	20:	// Oczekiwanie na zapis statusu - sprawdzenie wyniku
		IF stStationSettings.bSkipCheckStatusSaveResult THEN
			fbLogger.mAppendCurrentLine(bBreakLine := FALSE, sAddSep := '', sAppendText:= ', CSSR_Skiped');	
			IF bLastStatus THEN
				iCtr_PIM_PartsOK := iCtr_PIM_PartsOK +1;
			ELSE
				iCtr_PIM_PartsNOK := iCtr_PIM_PartsNOK +1;
			END_IF
			iWorkStep := 25;			
		ELSIF NOT bInsertStatus THEN
			IF bStatusSavedOK THEN
				IF bLastStatus THEN
					iCtr_PIM_PartsOK := iCtr_PIM_PartsOK +1;
				ELSE
					iCtr_PIM_PartsNOK := iCtr_PIM_PartsNOK +1;
				END_IF
				fbLogger.mAppendCurrentLine(bBreakLine := FALSE, sAddSep := '', sAppendText:= ', StatusSaved');
				iWorkStep := 25;	
			ELSE
				fbLogger.mAppendCurrentLine(bBreakLine := FALSE, sAddSep := '', sAppendText:= ', StatusNotSaved');
				mNewEvent(nInputErrorID := nPIM_ErrorCodes.StatusSaveError, nEventType := nPIM_EventClasses.Alarm, tMessageTime := T#0S);
			END_IF
		END_IF
		
	25:	// Oczekiwanie na zakończenie operacji
		IF NOT bSaveStatus THEN 
			fbLogger.mAppendCurrentLine(bBreakLine := TRUE, sAddSep := '', sAppendText:= ', OperEnded_BaseState_2');
			bNewOperationInProgress := FALSE;
			iWorkStep := 10;	
		END_IF

	99:
		IF stPimInOut.bConfirmEvent AND stPimInOut.bPIMActive THEN
			bResetSignal := TRUE;
			fbLogger.mAddLine(sTextToSave := CONCAT(STR1:= 'Reset bledu - wewnetrznego', STR2:= stPimInOut.sErrorCodePLC ) );
			IF 	nErrorID = nPIM_ErrorCodes.SelectStationIdError THEN 		// Błąd w inicjalizacji stanowiska do pracy
				nErrorID := nPIM_ErrorCodes.NoError;
				iWorkStep := 0;
			ELSIF nErrorID = nPIM_ErrorCodes.StatusSaveError THEN			// Gdy błąd zapisu statusu spróbuj jeszcze raz
				nErrorID := nPIM_ErrorCodes.NoError;
				bInsertStatus := TRUE;
				iWorkStep := 20;
			ELSE
				nErrorID := nPIM_ErrorCodes.NoError;
				iWorkStep := 0;
			END_IF
			IF nErrorID = nPIM_ErrorCodes.NoError THEN	// Jeśli błąd potwierdzony
				stPimInOut.bNonBlockingAlarm := stPimInOut.bAlarmPLC := stPimInOut.bWorkBlock_PLC := FALSE;
				stPimInOut.sErrorCodePLC := '';
				bResetSignal := FALSE;
				nEventType := nPIM_EventClasses.NoError;
			END_IF
		ELSIF nEventType = nPIM_EventClasses.Message THEN
				iWorkStep := 10;
		ELSE
			IF (nEventType <>nPIM_EventClasses.NoError) AND (NOT stPimInOut.bAlarmPLC AND NOT stPimInOut.bWorkBlock_PLC)  THEN
				mNewEvent(nInputErrorID := nPIM_ErrorCodes.UnKnownAlarm, nEventType := nPIM_EventClasses.Error, tMessageTime := T#0S);	
			END_IF
		END_IF
	
END_CASE

ACT_PimCmdsHandling();		// Obsługa komend z/do PIMu
ACT_SqlDataReturnCmd();		// Obsługa zapytań SQL do DB


// Automatyczne kasowanie wiadomości po zadanym czasie wyświetlania lub alarmu przy starcie nowej operacji
fbTON_MessageTimer();
IF stPimInOut.bNonBlockingAlarm AND (fbTON_MessageTimer.Q OR nMachineState = nPIM_MachineStates._3_NewOperationStarted) THEN
	fbTON_MessageTimer(IN:= FALSE);
	stPimInOut.sErrorCodePLC := '';
	stPimInOut.bNonBlockingAlarm := stPimInOut.bAlarmPLC := FALSE;
	nEventType := nPIM_EventClasses.NoError;
END_IF

fbTON_ServiceMessageTimer();		// Reset wiadomości serwisowej
IF fbTON_ServiceMessageTimer.Q THEN
	fbTON_ServiceMessageTimer(IN:= FALSE);
	stPimInOut.sPlcServiceMessage := '';
END_IF

IF GVL_Aircom.stAC_DT_Data.bNew_Shift OR bTestZapisu THEN
	iCtrMem_Operations := iCtr_Operations;
	iCtrMem_OperationsInterrupted := iCtr_OperationsInterrupted;
	iCtrMem_OperationsEndedOK := iCtr_OperationsEndedOK;
	iCtrMem_OperEndedOK_Method := iCtr_OperEndedOK_Method;
	iCtrMem_OperationsEndedNOK := iCtr_OperationsEndedNOK;
	iCtrMem_PIM_PartsOK := iCtr_PIM_PartsOK;
	iCtrMem_PIM_PartsNOK := iCtr_PIM_PartsNOK;
	iCtrMem_PIM_ReworkYes := iCtr_PIM_ReworkYes;
	iCtrMem_PIM_PartOK_SaveError := iCtr_PIM_PartOK_SaveError;
	iCtrMem_PIM_PartNOK_SaveError := iCtr_PIM_PartNOK_SaveError;
	iCtrMem_StatusSaveOK := iCtr_StatusSaveOK;
	iCtrMem_StatusSaveError := iCtr_StatusSaveError;
	iCtrMem_Errors := iCtr_Errors;
	iCtr_Operations:= iCtr_OperationsInterrupted:= iCtr_OperationsEndedOK:= iCtr_OperEndedOK_Method:= iCtr_OperationsEndedNOK:= 0; 
	iCtr_PIM_PartsOK:= iCtr_PIM_PartsNOK:= iCtr_PIM_ReworkYes:= iCtr_PIM_PartOK_SaveError := iCtr_PIM_PartNOK_SaveError:= iCtr_StatusSaveOK:= iCtr_StatusSaveError:= iCtr_Errors:= 0;

fbLogger.mAddLine(sTextToSave := CONCAT(STR1:= 'Nowa zmiana - ', STR2:= UINT_TO_STRING( GVL_Aircom.stAC_DT_Data.uiShiftNumber) ));
	fbLogger.mSaveBuffor();
	bTestZapisu := FALSE;
	bWriteHistoricData := TRUE;
END_IF
IF bWriteHistoricData AND fbLogger.bBufferEmpty THEN
		fbFormatStr(sFormat := 'PrevShiftReport: Oper-%d, OperInt-%d, OperOK-%d, OperOK_M-%d, OperNOK-%d',
		arg1 := F_INT(iCtrMem_Operations), 
		arg2 := F_INT(iCtrMem_OperationsInterrupted), 
		arg3 := F_INT(iCtrMem_OperationsEndedOK), 
		arg4 := F_INT(iCtrMem_OperEndedOK_Method), 
		arg5 := F_INT(iCtrMem_OperationsEndedNOK));  
	fbLogger.mAddLine(sTextToSave := fbFormatStr.sOut );
	fbFormatStr(sFormat := 'PrevShiftReport: PartsPIM_OK-%d, PartsPIM_NOK-%d, PartsPIM_ReworkYes-%d, PartsPIM_OK_missed-%d, PartsPIM_NOK_Missed-%d',
		arg1 := F_INT(iCtrMem_PIM_PartsOK), 
		arg2 := F_INT(iCtrMem_PIM_PartsNOK), 
		arg4 := F_INT(iCtrMem_PIM_ReworkYes),
		arg5 := F_INT(iCtrMem_PIM_PartOK_SaveError), 
		arg6 := F_INT(iCtrMem_PIM_PartNOK_SaveError));  
	fbLogger.mAddLine(sTextToSave := fbFormatStr.sOut );
	fbFormatStr(sFormat := 'PrevShiftReport: StatusSaveOK-%d, StatusSaveError-%d, Errors-%d, CmdReset- %d',
		arg1 := F_INT(iCtrMem_StatusSaveOK), 
		arg2 := F_INT(iCtrMem_StatusSaveError), 
		arg3 := F_INT(iCtrMem_Errors), 
		arg3 := F_UINT(in:=uiCtr_CmdReset));  
	uiCtr_CmdReset := 0;
	fbLogger.mAddLine(sTextToSave := fbFormatStr.sOut );	
	fbLogger.mSaveBuffor();
	bWriteHistoricData := FALSE;
END_IF

fbTON_ConfirmReset(IN:= stPimInOut.bConfirmEvent, PT:= T#3S);
stPimInOut.bConfirmEvent R= fbTON_ConfirmReset.Q;

PROPERTY PartsCtr_NOK : INT
GET
PartsCtr_NOK := iCtr_PIM_PartsNOK;
END_GET
END_PROPERTY

PROPERTY PartsCtr_OK : INT
GET
PartsCtr_OK := iCtr_PIM_PartsOK;
END_GET
END_PROPERTY

// The number of actually displayed error code ex "601"
PROPERTY prActiveErrorCode : STRING
GET
prActiveErrorCode := stPimInOut.sErrorCodePLC;
END_GET
END_PROPERTY

(* Get CMD Value from PIM*)
PROPERTY prCMD : STRING
GET
IF __ISVALIDREF(stPimInOut) THEN
	prCMD := sCmdToSendToMachine;
	sCmdToSendToMachine := '';	
END_IF
END_GET
END_PROPERTY

(* Get info *)
PROPERTY prCurrentMachineState : nPIM_MachineStates
GET
prCurrentMachineState := nMachineState;
END_GET
END_PROPERTY

(* Get info *)
PROPERTY prErrorClassExt : nPIM_EventClasses
GET
prErrorClassExt := nActEventClass;
END_GET
END_PROPERTY

(* Get info *)
PROPERTY prErrorConfirmActive : BOOL
GET
IF __ISVALIDREF(stPimInOut) THEN
	prErrorConfirmActive := stPimInOut.bConfirmEvent;
END_IF
END_GET
END_PROPERTY

(* Get info *)
PROPERTY prExternalEvtWaitInQueue : BOOL
GET
prExternalEvtWaitInQueue := FALSE;
END_GET
END_PROPERTY

(* Get info is PIM is active*)
PROPERTY prLastSavedStatus : BOOL
GET
prLastSavedStatus := bLastStatus;
END_GET
END_PROPERTY

(* Get info is PIM is active*)
PROPERTY prNokReportedSource : nPIM_ReportedNokSource
GET
prNokReportedSource := nReoprtedNokSource;
END_GET
END_PROPERTY

(* Get info is PIM is active*)
PROPERTY prOperEnded : BOOL
GET
prOperEnded := bOperationEnded;
END_GET
END_PROPERTY

(* Get info is PIM is active*)
PROPERTY prOperInProgress : BOOL
GET
prOperInProgress := nMachineState >= nPIM_MachineStates._3_NewOperationStarted AND nMachineState <= nPIM_MachineStates._6_ReturningToBaseState;
END_GET
END_PROPERTY

(* Get info is PIM is active*)
PROPERTY prPimActive : BOOL
GET
IF __ISVALIDREF(stPimInOut) THEN
	prPimActive := stPimInOut.bPIMActive;
END_IF
END_GET
END_PROPERTY

(* Get info *)
PROPERTY prPimBlockWork : BOOL
GET
IF __ISVALIDREF(stPimInOut) THEN
	prPimBlockWork := stPimInOut.bWorkBlock_PIM;
END_IF
END_GET
END_PROPERTY

(* Get info *)
PROPERTY prPlcBlockWork : BOOL
GET
IF __ISVALIDREF(stPimInOut) THEN
	prPlcBlockWork := stPimInOut.bWorkBlock_PLC;
END_IF
END_GET
END_PROPERTY

(* Get info is PIM is active*)
PROPERTY prReworkStatus : nPIM_ReworkSelect
GET
prReworkStatus := nReworkMenuStatus;
END_GET
END_PROPERTY

// Get info if station data is correctlly downloaded from database
PROPERTY prStationDataOK : BOOL
GET
prStationDataOK := bStationDataOK;
END_GET
END_PROPERTY

(* Get info is test mode is active*)
PROPERTY prTestMode : BOOL
GET
IF __ISVALIDREF(stPimInOut) THEN
	prTestMode := stPimInOut.bTestMode;
END_IF
END_GET
END_PROPERTY

(* Get info is user are logged?*)
PROPERTY prUserLogged : BOOL
GET
prUserLogged := fbTON_UserLogedDeleyed.Q;
END_GET
END_PROPERTY

(* Get info *)
PROPERTY prWorkPermission : BOOL
GET
IF __ISVALIDREF(stPimInOut) THEN
	prWorkPermission := stPimInOut.bTestMode OR NOT stPimInOut.bPIMActive OR (stPimInOut.bUSerLogged AND NOT stPimInOut.bWorkBlock_PIM AND NOT stPimInOut.bWorkBlock_PLC
					AND (NOT stPimInOut.bAlarmPLC OR stPimInOut.bNonBlockingAlarm) AND bMachineParamsOK AND bStationDataOK AND NOT bRetool AND NOT bMachParamsReadFromDB 
					AND NOT bMachParamsSendToDB);
END_IF
END_GET
END_PROPERTY

(* Get info is that machine is EOL*)
PROPERTY prIsEol : BOOL
GET
prIsEol := stRetDataLineStation.IsEOL;
END_GET
END_PROPERTY

(* Get Station name followed by machine number ex: 'CA01PL19_1'*)
PROPERTY prPartCodeNumber : STRING(250)
GET
prPartCodeNumber := stRetDataLineStation.PartCodeNumber;
END_GET
END_PROPERTY

(* Get Hidden status info*)
PROPERTY prIsHidden : BOOL
GET
prIsHidden := bIsHidden;
END_GET
END_PROPERTY

(* Get Line name ex: 'CA01PL'*)
PROPERTY prLineName : STRING(31)
GET
prLineName := sLineName;
END_GET
END_PROPERTY

(* Get Machine number*)
PROPERTY prMachNumber : INT
GET
prMachNumber := iMachineNumber;
END_GET
END_PROPERTY

(* Get Station name followed by machine number ex: 'CA01PL19_1'*)
PROPERTY prStationAlias : STRING(31)
GET
prStationAlias := CONCAT(STR1:= CONCAT(STR1:= sStationName, '_'), INT_TO_STRING(iMachineNumber));
END_GET
END_PROPERTY

(* Get Station name ex: 'CA01PL19'*)
PROPERTY prStationName : STRING(31)
GET
prStationName := sStationName;
END_GET
END_PROPERTY

// Zapis do DB dodatkowego kodu błędu - jeśli rozkaz dodany do kolejki zmienna wyjściowa ma wartość TRUE, jeśli nie (błąd dodania) FALSE
METHOD m_SqlInsAdditionalError : BOOL
VAR_INPUT
	sErrCode:STRING(10);		// Kod błędu do wysłania
END_VAR
VAR
	bResult:BOOL;
END_VAR
IF sErrCode <> '' AND stRetDataLineStation.IdStacji <> 0 THEN
	stSqlComandDataTMP.nCmdState:= nSQL_CmdExecState.New;
	stSqlComandDataTMP.nCmdType:=nSQL_CmdTypes.InsAdditionalError;
	stSqlComandDataTMP.bWaitForDataReturn:=FALSE;
	sFormat := 'INSERT INTO [dbo].[ProductionLineStationAdditionalError] (IdLineStation, MachineNumber, IdMachineError) VALUES (%d, %d, COALESCE( (SELECT Id FROM [dbo].[ProductionMachineError] WHERE Active = 1 AND Code = $'%s$'), -9223372036854775285))';
	fbFormatStr2(pFormatString := ADR(sFormat),
			arg1:= F_DINT(stRetDataLineStation.IdStacji),
			arg2:= F_INT(iMachineNumber),
			arg3:= F_STRINGEx(sErrCode),
			pDstString := ADR(stSqlComandDataTMP.sCmdExpression), nDstSize := SIZEOF(stSqlComandDataTMP.sCmdExpression));

	stSqlComandDataTMP.pReturnedData := 0;
	stSqlComandDataTMP.uiReturnedDataSize := 0;	
	IF I_SqlCore <> 0 THEN
		bResult := I_SqlCore.mAddCmdToQueue(ADR(stSqlComandDataTMP));
	END_IF
	m_SqlInsAdditionalError := bResult;
ELSE
	m_SqlInsAdditionalError := FALSE;
END_IF
END_METHOD

// Zapis do DB licznika zużycia powietrza - jeśli rozkaz dodany do kolejki zwraca TRUE, jeśli nie FALSE
METHOD m_SqlInsCompressedAirConsumption : BOOL
VAR_INPUT
	rActCompressedAirConsumption:REAL;		// Wartość licznika zużycia sprężonego powietrza
END_VAR
IF rActCompressedAirConsumption <> 0 AND stRetDataLineStation.IdLinii <> 0 THEN
	stSqlComandDataTMP.nCmdState:= nSQL_CmdExecState.New;
	stSqlComandDataTMP.nCmdType:=nSQL_CmdTypes.InsCompressedAirCons;
	stSqlComandDataTMP.bWaitForDataReturn:=FALSE;
	
	sFormat := 'INSERT INTO `ProductionConsumption_CompressedAir` (`IdLine`, `CounterValue`, `ValueUnit`) VALUES ( %d, %.3f, $'m3$')';
	fbFormatStr2(pFormatString := ADR(sFormat),
			arg1:= F_DINT(stRetDataLineStation.IdLinii),
			arg2:= F_REAL(rActCompressedAirConsumption),
			pDstString := ADR(stSqlComandDataTMP.sCmdExpression), nDstSize := SIZEOF(stSqlComandDataTMP.sCmdExpression));
	stSqlComandDataTMP.pReturnedData := 0;
	stSqlComandDataTMP.uiReturnedDataSize := 0;	
	IF I_SqlCore <> 0 THEN
		m_SqlInsCompressedAirConsumption := I_SqlCore.mAddCmdToQueue(ADR(stSqlComandDataTMP));
	END_IF	
ELSE
	m_SqlInsCompressedAirConsumption := FALSE;
END_IF
END_METHOD

// Zapis do DB relacji ostatniego statusu z kodem błędu - jeśli rozkaz dodany do kolejki zwraca TRUE, jeśli nie FALSE
METHOD m_SqlInsDefectRelation : BOOL
VAR_INPUT
	sErrCode:STRING(10);			// Kod błędu
END_VAR
IF sErrCode <> '' THEN
	stSqlComandDataTMP.nCmdState:= nSQL_CmdExecState.New;
	stSqlComandDataTMP.nCmdType:=nSQL_CmdTypes.InsDefectRelation;
	stSqlComandDataTMP.bWaitForDataReturn:=FALSE;
	
	sFormat := 'INSERT INTO [dbo].[ProductionMachinePartsStatusDefectRelation] (IdPartStatus, IdMachineError) values (%d, (SELECT Id FROM [dbo].[ProductionMachineError] WHERE Active = 1 AND Code = $'%s$'))';
	fbFormatStr2(pFormatString := ADR(sFormat),
			arg1:= F_LINT(liLPartStatusId),
			arg2:= F_STRINGEx(sErrCode),
			pDstString := ADR(stSqlComandDataTMP.sCmdExpression), nDstSize := SIZEOF(stSqlComandDataTMP.sCmdExpression));

	stSqlComandDataTMP.pReturnedData := 0;
	stSqlComandDataTMP.uiReturnedDataSize := 0;	
	IF I_SqlCore <> 0 THEN
		m_SqlInsDefectRelation := I_SqlCore.mAddCmdToQueue(ADR(stSqlComandDataTMP));
	END_IF
ELSE
	m_SqlInsDefectRelation := FALSE;
END_IF
END_METHOD

// Zapis do DB licznika zużycia energi na stanowisku - jeśli rozkaz dodany do kolejki zwraca TRUE, jeśli nie FALSE
METHOD m_SqlInsEnergyConsumption : BOOL
VAR_INPUT
	rActEnergyConsumption:REAL;			// Wartość licznika zużycia energii elektrycznej
END_VAR
IF rActEnergyConsumption <> 0 AND stRetDataLineStation.IdStacji <> 0 THEN
	stSqlComandDataTMP.nCmdState:= nSQL_CmdExecState.New;
	stSqlComandDataTMP.nCmdType:=nSQL_CmdTypes.InsEnergyCons;
	stSqlComandDataTMP.bWaitForDataReturn:=FALSE;
	
	sFormat := 'INSERT INTO `ProductionConsumption_Energy` (`IdLineStation`, `CounterValue`, `ValueUnit`) VALUES ( %d, %.3f, $'kWh$')';
	fbFormatStr2(pFormatString := ADR(sFormat),
			arg1:= F_DINT(stRetDataLineStation.IdStacji),
			arg2:= F_REAL(rActEnergyConsumption),
			pDstString := ADR(stSqlComandDataTMP.sCmdExpression), nDstSize := SIZEOF(stSqlComandDataTMP.sCmdExpression));

	stSqlComandDataTMP.pReturnedData := 0;
	stSqlComandDataTMP.uiReturnedDataSize := 0;	
	IF I_SqlCore <> 0 THEN
		m_SqlInsEnergyConsumption := I_SqlCore.mAddCmdToQueue(ADR(stSqlComandDataTMP));
	END_IF
ELSE
	m_SqlInsEnergyConsumption := FALSE;
END_IF
END_METHOD

// Zapis do DB danych rozszerzonych operacji - jeśli rozkaz dodany do kolejki zwraca TRUE, jeśli nie FALSE
METHOD m_SqlInsertExtendedData : BOOL		
VAR_INPUT
	pParameters: POINTER TO BYTE;				// Wskaźnik na tablicę elementów typu PIM_ExtDataRow
	uiArraySize: UINT;							// Rozmiar tablicy parametrów (może być pojedyncza zmienna)
END_VAR
VAR
	pExtData: POINTER TO stPIM_ExtDataRow;
	i:UINT;
	uiLastIndex:UINT;
END_VAR
uiLastIndex := uiArraySize/ SIZEOF(stPIM_ExtDataRow);
IF pParameters <> 0 AND uiArraySize > 0 AND uiLastIndex > 0 AND liLPartStatusId <> 0 THEN		// Zabezpieczenie przed brakiem danych wejściowych
	stSqlComandDataTMP.sCmdExpression := 'INSERT INTO `ProductionMachinePartParams` (`IdPartStatus`,`Name`,`Value`) VALUES';
	pExtData := pParameters;
	FOR i:=1 TO uiLastIndex DO		// Dodanie do stringa wartości
		IF i = uiLastIndex THEN		// Ostatnia wartość bez przecinka
			fbFormatStr(sFormat:= ' (%d,$'%s$',$'%s$')',arg1 := F_LINT(in:=liLPartStatusId), arg2 := F_STRINGEx(pExtData^.sName), arg3 := F_STRINGEx(pExtData^.sValue));
		ELSE
			fbFormatStr(sFormat:= ' (%d,$'%s$',$'%s$'),',arg1 := F_LINT(in:=liLPartStatusId), arg2 := F_STRINGEx(pExtData^.sName), arg3 := F_STRINGEx(pExtData^.sValue));		
			pExtData := pExtData + SIZEOF(stPIM_ExtDataRow);		// Przejście na kolejny indeks w tablicy
		END_IF
		CONCAT2(pSrcString1 := ADR(stSqlComandDataTMP.sCmdExpression), pSrcString2 := ADR(fbFormatStr.sOut), pDstString := ADR(stSqlComandDataTMP.sCmdExpression), nDstSize:= SIZEOF(stSqlComandDataTMP.sCmdExpression));
	END_FOR
	stSqlComandDataTMP.nCmdState:= nSQL_CmdExecState.New;
	stSqlComandDataTMP.nCmdType:=nSQL_CmdTypes.InsExtendedData;
	stSqlComandDataTMP.bWaitForDataReturn:=FALSE;
	stSqlComandDataTMP.pReturnedData := 0;
	stSqlComandDataTMP.uiReturnedDataSize := 0;
	IF I_SqlCore <> 0 THEN
  		m_SqlInsertExtendedData := I_SqlCore.mAddCmdToQueue(ADR(stSqlComandDataTMP));
	END_IF
ELSE
	m_SqlInsertExtendedData := FALSE;
END_IF
END_METHOD

// Zapis do DB parametrów maszyny przypisanych do aktualnego komponentu - gdy rozkaz zostanie wykonany zwraca TRUE
METHOD m_SqlInsMachineParamsData : BOOL
VAR_INPUT
	pParamsData: POINTER TO BYTE;		// Wskaźnik do bloku parametrów maszyny
	uiParamsDataSize: UINT;				// ROzmiar bloku danych parametrów maszyny
	wCrcSumOfParameters:WORD:= 0;
END_VAR
VAR_OUTPUT
	bProcessing:BOOL;					// Przetwarzanie rozkazu trwa (rozkaz dodany do kolejki)
	bResultOK:BOOL;						// Wynik wykonania rozkazu (do sprawdzenia gdy metoda zwróci TRUE)
	diParamsId:DINT;					// Id parametrów w DB
END_VAR
VAR
	sStringTMP:STRING(1000);
	iCRC16sum: INT;
END_VAR

// Sprawdzenie danych wejściowych - jeśli błędne przerwij procedure
IF pParamsData = 0 OR uiParamsDataSize = 0 OR stRetDataLineStation.IdStacji = 0 THEN 
	nErrorID:=nPIM_ErrorCodes.ProgramError;
	RETURN;
END_IF

// Rezerwacja struktury danych dla zapytania
IF NOT bReturnDataBusy OR bReturnDataReserved_InsMachParams THEN
	IF NOT bCmdSended THEN	// Przygotowanie danych do zapytania
		stSqlComandData.nCmdState:= nSQL_CmdExecState.New;
		stSqlComandData.nCmdType:=nSQL_CmdTypes.InsMachineParams;
		stSqlComandData.byExecutingNodeNb:=0;
		stSqlComandData.bWaitForDataReturn:=TRUE;
		
		IF wCrcSumOfParameters <> 0 THEN
			iCRC16sum := WORD_TO_INT(wCrcSumOfParameters);
		ELSE
			iCRC16sum := WORD_TO_INT(F_DATA_TO_CRC16_CCITT(pData := pParamsData, cbData := uiParamsDataSize, crc:= 0));
		END_IF
		
		sFormat := 'UPDATE [dbo].[ProductionMachineParameters] SET Active = 0 WHERE IdLineStation = %d AND MachineNumber = %d AND IdComposedPart = %d DECLARE @ID_INSERTED TABLE (Id INT) INSERT INTO [dbo].[ProductionMachineParameters] 
					(IdLineStation, MachineNumber, IdComposedPart,ParamsData,CRC_Sum,ParamsSizeInBytes) OUTPUT INSERTED.ID INTO @ID_INSERTED VALUES (%d, %d, %d, CAST(';
		fbFormatStr2(pFormatString := ADR(sFormat),
			arg1:= F_DINT(stRetDataLineStation.IdStacji),
			arg2:= F_INT(iMachineNumber),
			arg3:= F_LINT(stRetDataLineStation.IdOutComposedPart),
			arg4:= F_DINT(stRetDataLineStation.IdStacji),
			arg5:= F_INT(iMachineNumber),
			arg6:= F_LINT(stRetDataLineStation.IdOutComposedPart),
			pDstString := ADR(stSqlComandData.sCmdExpression), nDstSize := SIZEOF(stSqlComandData.sCmdExpression));
			
		sFormat := ' AS VARBINARY(%d)), %d,%d) SELECT Id FROM @ID_INSERTED';
		fbFormatStr2(pFormatString := ADR(sFormat),
			arg1:= F_UINT(uiParamsDataSize),
			arg2:= F_INT(iCRC16sum),
			arg3:= F_UINT(uiParamsDataSize),
			pDstString := ADR(sStringTMP), nDstSize := SIZEOF(sStringTMP));

		
//		stDBCmdData.sCmdExpression := 'DECLARE @ID_INSERTED TABLE (Id INT) INSERT INTO ProductionMachineParameters (IdLineStation, MachineNumber, IdComposedPart, ParamsData, CRC_Sum) OUTPUT INSERTED.ID INTO @ID_INSERTED VALUES ({IdLineStation}, {MachineNumber}, {IdComposedPart}, ( CONVERT ( VARBINARY({iStructDataSize}), {astStructRawData}) ), {iCRC16sum}) SELECT Id FROM @ID_INSERTED';
//		stDBCmdData.sCmdExpression := 'DECLARE @ID_INSERTED TABLE (Id INT) INSERT INTO ProductionMachineParameters (IdLineStation, MachineNumber, IdComposedPart, ParamsData, CRC_Sum) OUTPUT INSERTED.ID INTO @ID_INSERTED VALUES ({IdLineStation}, {MachineNumber}, (SELECT IdOutComposedPart FROM ProductionLineStation WHERE Id ={IdLineStation}), {astStructRawData}, {iCRC16sum}) SELECT Id FROM @ID_INSERTED';
//		stDBCmdData.sCmdExpression := 'DECLARE @ID_INSERTED TABLE (Id INT) INSERT INTO ProductionMachineParameters (IdLineStation, MachineNumber, IdComposedPart, ParamsData, CRC_Sum) OUTPUT INSERTED.ID INTO @ID_INSERTED VALUES ({IdLineStation}, {MachineNumber}, (SELECT IdOutComposedPart FROM ProductionLineStation WHERE Id ={IdLineStation}), CAST({astStructRawData} AS VARBINARY({iStructDataSize})), {iCRC16sum}) SELECT Id FROM @ID_INSERTED';
//		stDBCmdData.sCmdExpression := 'DECLARE @ID_INSERTED TABLE (Id INT) INSERT INTO ProductionMachineParameters (IdLineStation, MachineNumber, IdComposedPart, ParamsData, CRC_Sum) OUTPUT INSERTED.ID INTO @ID_INSERTED VALUES ({IdLineStation}, {MachineNumber}, {IdComposedPart}, {astStructRawData}, {iCRC16sum}) SELECT Id FROM @ID_INSERTED';
//		stDBCmdData.sCmdExpression := 'DECLARE @ID_INSERTED TABLE (Id INT) INSERT INTO ProductionMachineParameters (IdLineStation, MachineNumber, IdComposedPart, ParamsData, CRC_Sum) OUTPUT INSERTED.ID INTO @ID_INSERTED VALUES ({IdLineStation}, {MachineNumber}, {IdComposedPart}, CAST({astStructRawData} AS VARBINARY({iStructDataSize})), {iCRC16sum}) SELECT Id FROM @ID_INSERTED';
//		stDBCmdData.sCmdExpression := 'UPDATE [dbo].[ProductionMachineParameters] SET Active = 0 WHERE IdLineStation = {IdLineStation} AND IdComposedPart = {IdComposedPart} DECLARE @ID_INSERTED TABLE (Id INT) INSERT INTO [dbo].[ProductionMachineParameters] (IdLineStation, MachineNumber, IdComposedPart,ParamsData,CRC_Sum,ParamsSizeInBytes) OUTPUT INSERTED.ID INTO @ID_INSERTED VALUES ({IdLineStation}, {MachineNumber}, {IdComposedPart}), CAST( {astStructRawData} AS VARBINARY(';
		stSqlComandData.sCmdExpression := 'UPDATE [dbo].[ProductionMachineParameters] SET Active = 0 WHERE IdLineStation = {IdLineStation} AND MachineNumber = {MachineNumber} AND IdComposedPart = {IdComposedPart} DECLARE @ID_INSERTED TABLE (Id INT) INSERT INTO [dbo].[ProductionMachineParameters] (IdLineStation, MachineNumber, IdComposedPart,ParamsData,CRC_Sum,ParamsSizeInBytes) OUTPUT INSERTED.ID INTO @ID_INSERTED VALUES ({IdLineStation}, {MachineNumber}, {IdComposedPart}, CAST( {astStructRawData} AS VARBINARY(';
		sStringTMP := UINT_TO_STRING(uiParamsDataSize);
		CONCAT2(pSrcString1 := ADR(stSqlComandData.sCmdExpression), pSrcString2 := ADR(sStringTMP),pDstString := ADR(stSqlComandData.sCmdExpression), nDstSize := SIZEOF(stSqlComandData.sCmdExpression));
		sStringTMP := ')), {iCRC16sum},{iStructDataSize}) SELECT Id FROM @ID_INSERTED';
		CONCAT2(pSrcString1 := ADR(stSqlComandData.sCmdExpression),pSrcString2 := ADR(sStringTMP),pDstString := ADR(stSqlComandData.sCmdExpression), nDstSize := SIZEOF(stSqlComandData.sCmdExpression));
		
		stSqlComandData.pReturnedData := ADR(diMachineParamsInsertId);
		stSqlComandData.uiReturnedDataSize := SIZEOF(diMachineParamsInsertId);
		stSqlComandData.bSQL_OK := stSqlComandData.bSQL_Done := FALSE;
		// Próba dodania komendy do kolejki
		IF I_SqlCore <> 0 AND_THEN I_SqlCore.mAddCmdToQueue(ADR(stSqlComandData)) THEN
			bCmdSended := bReturnDataBusy := bReturnDataReserved_InsMachParams := TRUE;		// Zajęcie struktury danych
			diMachineParamsInsertId := 0;
		ELSE
			bResultOk := FALSE;
			nErrorID:=nPIM_ErrorCodes.ParamsSaveToDB_Error;
			m_SqlInsMachineParamsData := bCmdAddError := TRUE;
		END_IF
	ELSIF stSqlComandData.bSQL_Done THEN
		IF stSqlComandData.bSQL_OK THEN
			diParamsId := diMachineParamsInsertId;
		ELSE
			nErrorID:=nPIM_ErrorCodes.ParamsSaveToDB_Error;
		END_IF
		bInsMachineParamsData := TRUE;	// Odśwież parametrów w strukturze PIM, skasowanie zmiennej bCmdSended
		bResultOK := stSqlComandData.bSQL_OK;
		m_SqlInsMachineParamsData := bUpdateData := TRUE;
	END_IF
END_IF
bProcessing := bCmdSended AND NOT stSqlComandData.bSQL_Done;
END_METHOD

// Zapis do DB statusu ostatniej operacji - gdy rozkaz zostanie wykonany zwraca TRUE
METHOD m_SqlSelInsStatus : BOOL
VAR_INPUT
	bStatus:BOOL:= FALSE;		// Status operacji do zapisania
	sErrCode:STRING(10);		// kod błędu - tylko jeśli status  FALSE
	bSustein:BOOL:= FALSE;		// Jeśli TRUE po wywołaniu przez FbMaszyny wykonwyanie rozkazu przerzucone na fbStation (wysyłanie rozkazu w tle)- ustawiana odpowiednia flaga 
END_VAR
VAR_OUTPUT
	bProcessing:BOOL;			// Przetwarzanie rozkazu trwa (rozkaz dodany do kolejki)
	bResultOK:BOOL;				// Wynik wykonania rozkazu (do sprawdzenia gdy metoda zwróci TRUE)
	liStatusId:LINT;			// Id statusu części w DB
END_VAR

VAR
	byStatus: BYTE;
	byIsHidden: BYTE;
END_VAR
// Rezerwacja struktury danych dla zapytania
IF NOT bReturnDataBusy OR bReturnDataReserved_InsOperStat AND bStationIdValid THEN
	IF NOT bCmdSended THEN	// Przygotowanie danych do zapytania
		stSqlComandData.nCmdState:= nSQL_CmdExecState.New;
		stSqlComandData.nCmdType:=nSQL_CmdTypes.SelInsStatusOfOperation;
		stSqlComandData.byExecutingNodeNb:=0;
		stSqlComandData.bWaitForDataReturn:=TRUE;
		
		stSqlComandData.stStatusSaveParams.didLineStation := stRetDataLineStation.IdStacji;
		stSqlComandData.stStatusSaveParams.byStatus := BOOL_TO_BYTE(bStatus);
		IF bStatus THEN
			stSqlComandData.stStatusSaveParams.byIsHidden := BOOL_TO_BYTE(bIsHidden);
		ELSE
			stSqlComandData.stStatusSaveParams.byIsHidden := 0;
		END_IF
		stSqlComandData.stStatusSaveParams.byIsTestMode := BOOL_TO_BYTE(stPimInOut.bTestMode);
		stSqlComandData.stStatusSaveParams.iMachineNb := iMachineNumber;
		stSqlComandData.stStatusSaveParams.lrQuantity := 1.0;
		byStatus := BOOL_TO_BYTE(bStatus);
		byIsHidden := BOOL_TO_BYTE(bIsHidden);	
(*		IF bStatus THEN
			sFormat := 'DECLARE @ID_TABLE TABLE (Id bigint) insert into [dbo].[ProductionMachinePartsStatuses] (IdLineStation, Status, MachineNumber, IsHidden) output inserted.id into @ID_TABLE values (%d, %d, %d, %d) SELECT Top(1) Id FROM @ID_TABLE';
				fbFormatStr2(pFormatString := ADR(sFormat),
				arg1:= F_DINT(stRetDataLineStation.IdStacji),
				arg2:= F_BYTE(byStatus),
				arg3:= F_INT(iMachineNumber),
				arg4:= F_BYTE(byIsHidden),
				pDstString := ADR(stSqlComandData.sCmdExpression), nDstSize := SIZEOF(stSqlComandData.sCmdExpression));
		ELSE
			sFormat := 'DECLARE @ID_TABLE TABLE (Id bigint) insert into [dbo].[ProductionMachinePartsStatuses] (IdLineStation, Status, MachineNumber, IsHidden) output inserted.id into @ID_TABLE values (%d, %d, %d, %d) DECLARE @statusId bigint = (SELECT Top(1) Id FROM @ID_TABLE) INSERT INTO [dbo].[ProductionMachinePartsStatusDefectRelation] (IdPartStatus, IdMachineError) values (@statusId, (SELECT Id FROM [dbo].[ProductionMachineError] WHERE Active = 1 AND Code = $'%s$')) SELECT @statusId';
				fbFormatStr2(pFormatString := ADR(sFormat),
				arg1:= F_DINT(stRetDataLineStation.IdStacji),
				arg2:= F_BYTE(byStatus),
				arg3:= F_INT(iMachineNumber),
				arg4:= F_BYTE(byIsHidden),
				arg5:= F_STRINGEx(sErrCode),
				pDstString := ADR(stSqlComandData.sCmdExpression), nDstSize := SIZEOF(stSqlComandData.sCmdExpression));
		END_IF
*)
		bLastStatus := bStatus;
		sLastErrCode:= sErrCode;
		stSqlComandData.pReturnedData := ADR(liLPartStatusId);
		stSqlComandData.uiReturnedDataSize := SIZEOF(liLPartStatusId);
		bStatusSavedOK := stSqlComandData.bSQL_OK := stSqlComandData.bSQL_Done := FALSE;
		// Próba dodania komendy do kolejki
		IF I_SqlCore <> 0 AND_THEN I_SqlCore.mAddCmdToQueue(ADR(stSqlComandData)) THEN
			bCmdSended := bReturnDataBusy := bReturnDataReserved_InsOperStat := TRUE;		// Zajęcie struktury danych
			liLPartStatusId := 0;
			bInsertStatus S= bSustein;
		ELSE
			bResultOk := FALSE;
			m_SqlSelInsStatus := bCmdAddError := TRUE;
		END_IF
	ELSIF stSqlComandData.bSQL_Done THEN
		IF stSqlComandData.bSQL_OK THEN
			liStatusId := liLPartStatusId;	// Uaktualnij zmienną wyjściową
		END_IF
		bInsertStatus := TRUE;	// Odśwież parametrów w strukturze PIM, skasowanie zmiennej bCmdSended
		bResultOK := stSqlComandData.bSQL_OK;
		m_SqlSelInsStatus := bUpdateData := TRUE;
	END_IF
END_IF
bProcessing := bCmdSended AND NOT stSqlComandData.bSQL_Done;
END_METHOD

// Pobranie z DB statusu ostatniej operacji dla danego DM z poprzedniego stanowiska - gdy rozkaz zostanie wykonany zwraca TRUE
METHOD m_SqlSelLastOperationStatus : BOOL
VAR_INPUT
	sCodeDM:STRING(255);		// Identyfikator części (kod DataMatrix)
END_VAR
VAR_OUTPUT
	bProcessing:BOOL;			// Przetwarzanie rozkazu trwa (rozkaz dodany do kolejki)
	bResultOK:BOOL;				// Wynik wykonania rozkazu (do sprawdzenia gdy metoda zwróci TRUE)
	bPrevOperStat:BOOL;			// Status ostatniej operacji na poprzednim stanowisku
END_VAR
// Rezerwacja struktury danych dla zapytania
IF NOT bReturnDataBusy OR bReturnDataReserved_SelLastOperStat THEN
	IF NOT bCmdSended THEN
		// Przygotowanie danych do zapytania
		stSqlComandData.nCmdState:= nSQL_CmdExecState.New;
		stSqlComandData.nCmdType:=nSQL_CmdTypes.SelLastOperationStatus;
		stSqlComandData.byExecutingNodeNb:=0;
		stSqlComandData.bWaitForDataReturn:=TRUE;
		sFormat := 'SELECT TOP(1) PMPS.Status FROM [dbo].[ProductionMachinePartsStatuses] PMPS INNER JOIN [dbo].[ProductionLineStation] PLS ON PLS.Id = PMPS.IdLineStation WHERE PLS.Active = 1 AND PMPS.NumberId = $'%s$' AND PLS.Name = $'%s$' AND PMPS.IsHidden = 0 ORDER BY PMPS.Date desc';
		fbFormatStr2(pFormatString := ADR(sFormat),
			arg1:= F_STRINGEx(sCodeDM),
			arg2:= F_STRINGEx(sPrevStationName),
			pDstString := ADR(stSqlComandData.sCmdExpression), nDstSize := SIZEOF(stSqlComandData.sCmdExpression));
		stSqlComandData.pReturnedData := ADR(bPreviousOperationStatus);
		stSqlComandData.uiReturnedDataSize := SIZEOF(bPreviousOperationStatus);
		stSqlComandData.bSQL_OK := stSqlComandData.bSQL_Done := FALSE;
		// Próba dodania komendy do kolejki
		IF I_SqlCore <> 0 AND_THEN I_SqlCore.mAddCmdToQueue(ADR(stSqlComandData)) THEN
			bCmdSended := 	bReturnDataBusy := bReturnDataReserved_SelLastOperStat := TRUE;		// Zajęcie struktury danych
			bPreviousOperationStatus := FALSE;
		ELSE
			bResultOk := FALSE;
			m_SqlSelLastOperationStatus := bCmdAddError := TRUE;
		END_IF
	ELSIF stSqlComandData.bSQL_Done THEN		// Komenda została wykonana, sprawdzenie rezultatu
		IF stSqlComandData.bSQL_OK THEN
			bPrevOperStat := bPreviousOperationStatus;	// Uaktualnij zmienną wyjściową
		END_IF
		bSelPreviousStatus := TRUE;	// Odśwież parametrów w strukturze PIM, skasowanie zmiennej bCmdSended
		bResultOK := stSqlComandData.bSQL_OK;
		m_SqlSelLastOperationStatus := bUpdateData := TRUE;
	END_IF
END_IF
bProcessing := bCmdSended AND NOT stSqlComandData.bSQL_Done;
END_METHOD

// Pobranie z DB ID stanowiska - gdy rozkaz zostanie wykonany zwraca TRUE
METHOD PRIVATE m_SqlSelLineStationId : BOOL
VAR_INPUT
END_VAR
VAR_OUTPUT
	bProcessing:BOOL;			// Przetwarzanie rozkazu trwa (rozkaz dodany do kolejki)
	bResultOK:BOOL;				// Wynik wykonania rozkazu (do sprawdzenia gdy metoda zwróci TRUE)
	diStationId:DINT;			// Identyfikator stanowiska
	liIdCompossedPart:LINT;		// Identyfikator części wyjściowej
	bAutoSaveErrors:BOOL;		// Auto zapis błędów
	bAutoControlMachineParams:BOOL;		// Kontrola parametrów maszyny
	wCrcSumInDB:WORD;			// Suma CRC aktualnych parametrów maszyny dla złożenia wyjściowego
END_VAR
// Rezerwacja struktury danych dla zapytania
IF NOT bReturnDataBusy OR bReturnDataReserved_StationId THEN
	bStationIdValid := FALSE;
	IF NOT bCmdSended THEN
		// Przygotowanie danych do zapytania
		stSqlComandData.nCmdState:= nSQL_CmdExecState.New;
		stSqlComandData.nCmdType:=nSQL_CmdTypes.SelStationId;
		stSqlComandData.byExecutingNodeNb:=0;
		stSqlComandData.bWaitForDataReturn:=TRUE;
		sFormat := 'SELECT PL.Id, PLS.Id, PLS.IsAutoSaveErrors, PLS.IsEol, PLS.IdOutComposedPart, PMP.CRC_Sum, PCP.CodeNumber FROM [dbo].[ProductionLineStation] PLS INNER JOIN [dbo].[ProductionLine] PL on PLS.IdLine=PL.Id LEFT JOIN [dbo].[ProductionMachineParameters] PMP on PLS.Id=PMP.IdLineStation AND PLS.IdOutComposedPart=PMP.IdComposedPart AND PMP.MachineNumber=%d AND PMP.Active=1 LEFT JOIN [dbo].[ProductionComposedPart] PCP on PLS.IdOutComposedPart=PCP.Id AND PCP.Active=1 WHERE PL.Active = 1 AND PL.Name = $'%s$' AND PLS.Name = $'%s$' AND PLS.Active=1';
		fbFormatStr2(pFormatString := ADR(sFormat),
			arg1:= F_INT(iMachineNumber),
			arg2:= F_STRINGEx(sLineName),
			arg3:= F_STRINGEx(sStationName),
			pDstString := ADR(stSqlComandData.sCmdExpression), nDstSize := SIZEOF(stSqlComandData.sCmdExpression));
		stSqlComandData.pReturnedData := ADR(stRetDataLineStation);
		stSqlComandData.uiReturnedDataSize := SIZEOF(stRetDataLineStation);
		stSqlComandData.bSQL_OK := stSqlComandData.bSQL_Done := FALSE;
		// Próba dodania komendy do kolejki
		IF I_SqlCore <> 0 AND_THEN I_SqlCore.mAddCmdToQueue(ADR(stSqlComandData)) THEN
			bSelectStationId := bCmdSended := bReturnDataBusy := bReturnDataReserved_StationId := TRUE;		// Zajęcie struktury danych
			diStationId := 0;
			MEMSET(destAddr := ADR(stRetDataLineStation), n := SIZEOF(stRetDataLineStation), fillByte:= 0);		// Czyszczenie danych 
		ELSE
			bResultOk := FALSE;
			m_SqlSelLineStationId := bCmdAddError := TRUE;
		END_IF
	ELSIF stSqlComandData.bSQL_Done THEN
		IF stSqlComandData.bSQL_OK THEN
			diStationId := stRetDataLineStation.IdStacji;	// Uaktualnij zmienne wyjściowe
			liIdCompossedPart := stRetDataLineStation.IdOutComposedPart;
			bAutoSaveErrors := stRetDataLineStation.AutoSaveErrors;
			bAutoControlMachineParams := FALSE;// stRetDataLineStation.AutoControlMachineParams; 
			wCrcSumInDB:= stRetDataLineStation.CrcSumOfParams;
		END_IF
		bSelectStationId := bUpdateData := TRUE;	// Odświeżenie parametrów w strukturze PIM w cżęści głównej bloku funkcyjnego, skasowanie zmiennej bCmdSended
		bResultOK := stSqlComandData.bSQL_OK;
		m_SqlSelLineStationId := TRUE;
	END_IF
END_IF
bProcessing := bCmdSended AND NOT stSqlComandData.bSQL_Done;
END_METHOD

// Pobranie z DB sumy CRC parametrów pracy maszyny - gdy rozkaz zostanie wykonany zwraca TRUE
METHOD PRIVATE m_SqlSelMachineParamsCRC : BOOL
VAR_INPUT
	liIdCompossedPart:LINT;		// Identyfikator części wyjściowej dla którego powinna zostać pobrana suma 
END_VAR
VAR_OUTPUT
	bProcessing:BOOL;		// Przetwarzanie rozkazu trwa (rozkaz dodany do kolejki)
	bResultOK:BOOL;			// Wynik wykonania rozkazu (do sprawdzenia gdy metoda zwróci TRUE)
	diStationId:DINT;		// Identyfikator stanowiska
	wCrcFromDb:WORD;		// Suma CRC pobrana z DB
END_VAR
// Sprawdzenie danych wejściowych - jeśli błędne przerwij procedure
IF liIdCompossedPart = 0 OR stRetDataLineStation.IdStacji = 0 THEN
	m_SqlSelMachineParamsCRC := TRUE;
	bResultOK := FALSE;
	RETURN;
END_IF

// Rezerwacja struktury danych dla zapytania
IF NOT bReturnDataBusy OR bReturnDataReserved_SelMachParamsCRC THEN
	IF NOT bCmdSended THEN
		// Przygotowanie danych do zapytania
		stSqlComandData.nCmdState:= nSQL_CmdExecState.New;
		stSqlComandData.nCmdType:=nSQL_CmdTypes.SelMachineParamsCRC;
		stSqlComandData.byExecutingNodeNb:=0;
		stSqlComandData.bWaitForDataReturn:=TRUE;
	
		
		sFormat := 'SELECT CRC_Sum, FROM [dbo].[ProductionMachineParameters] WHERE Active = 1 AND IdLineStation = %d AND MachineNumber = %d AND IdComposedPart = %d';
		fbFormatStr2(pFormatString := ADR(sFormat),
			arg1:= F_DINT(stRetDataLineStation.IdStacji),
			arg2:= F_INT(iMachineNumber),
			arg3:= F_LINT(stRetDataLineStation.IdOutComposedPart),
			pDstString := ADR(stSqlComandData.sCmdExpression), nDstSize := SIZEOF(stSqlComandData.sCmdExpression));

(*		stSqlComandData.sCmdExpression := 'SELECT CRC_Sum, FROM [dbo].[ProductionMachineParameters] WHERE Active = 1 AND IdLineStation = {IdLineStation} AND MachineNumber = {MachineNumber} AND IdComposedPart = {IdComposedPart}';
		stSqlComandData.stCmdData.IdLineStation := stRetDataLineStation.IdStacji;
		stSqlComandData.stCmdData.MachineNumber := iMachineNumber;
		IF liIdCompossedPart = 0 THEN			// Jeśli 0 pobiera dla aktualnie produkowanego, można też pobrać dla konkretnego Id
			stSqlComandData.stCmdData.IdComposedPart := stRetDataLineStation.IdOutComposedPart;
		ELSE
			stSqlComandData.stCmdData.IdComposedPart := liIdCompossedPart;
		END_IF	*)
		stSqlComandData.pReturnedData := ADR(wCrcSumInDb);
		stSqlComandData.uiReturnedDataSize := SIZEOF(wCrcSumInDb);
		stSqlComandData.bSQL_OK := stSqlComandData.bSQL_Done := FALSE;
		// Próba dodania komendy do kolejki
		IF I_SqlCore <> 0 AND_THEN I_SqlCore.mAddCmdToQueue(ADR(stSqlComandData)) THEN
			bCmdSended := bReturnDataBusy := bReturnDataReserved_SelMachParamsCRC := TRUE;		// Zajęcie struktury danych
			wCrcSumInDb := 0;
		ELSE
			bResultOk := FALSE;
			m_SqlSelMachineParamsCRC := bCmdAddError := TRUE;
		END_IF
	ELSIF stSqlComandData.bSQL_Done THEN
		IF stSqlComandData.bSQL_OK THEN
			wCrcFromDb := wCrcSumInDb;	// Uaktualnij zmienne wyjściowe
		END_IF
		m_SqlSelMachineParamsCRC := TRUE;	// Odświeżenie parametrów w strukturze PIM w cżęści głównej bloku funkcyjnego, skasowanie zmiennej bCmdSended
		bResultOK := stSqlComandData.bSQL_OK;
		m_SqlSelMachineParamsCRC := bUpdateData := TRUE;
	END_IF
END_IF
bProcessing := bCmdSended AND NOT stSqlComandData.bSQL_Done;
END_METHOD

// Pobranie z DB parametrów pracy maszyny - gdy rozkaz zostanie wykonany zwraca TRUE
METHOD m_SqlSelMachineParamsData : BOOL
VAR_INPUT
	diParamsId:DINT:=0;				// Jeśli 0 - pobiera parametry dla aktualnego złożenia, jeśli <>0 wtedy pobiera zestaw parametrów o danym Id
	pParamsData:POINTER TO BYTE;	// Wskaźnik do struktury parametrów maszyny
	uiParamsDataSize:UINT;			// Rozmiar struktury danych parametrów maszyny
END_VAR
VAR_OUTPUT
	bProcessing:BOOL;				// Przetwarzanie rozkazu trwa (rozkaz dodany do kolejki)
	bResultOK:BOOL;					// Wynik wykonania rozkazu (do sprawdzenia gdy metoda zwróci TRUE)
	bNoMatchingParams:BOOL;			// Błąd - brak pasujących parametrów w DB
	bParametersUpdated:BOOL;		// Parametry maszyny uaktualnione
//	pParamsData: POINTER TO BYTE;
END_VAR
(*
Zapis i odczyt parametrów kontroluje blok klienta PIM, struktura w bloku przechowywana jest jako wskaźnik więc nie jest konieczne powiązanie ze strukturą parametrów maszyny.
Metoda pobiera z DB najnowszy zestaw parametrów lub zestaw o danym Id (jeśli Id nie jest równe 0), sprawdza czy rozmiary oraz suma CRC są zgodne - jeśli są przepisuje pobrane dane do wskaźnika wejściowego.
Jeśli nie co zrobić - może pytanie do użytkownika (przez komendy PIM) "Rozmiar/wartość danych niezgodna - pomiń lub nadpisz" - użytkownik wybierze odpowiendią opcje która zostanie zwrócona do PLC.
Póki co następuje automatyczne przepisanie niekompletnych lub niezgodnych parametrów.
*)

// Sprawdzenie danych wejściowych - jeśli błędne przerwij procedure
IF pParamsData = 0 OR uiParamsDataSize = 0 OR SEL(diParamsId=0, stRetDataLineStation.IdStacji = 0, stRetDataLineStation.IdStacji = 0 OR stRetDataLineStation.IdOutComposedPart = 0) THEN
	m_SqlSelMachineParamsData := TRUE;
	bResultOK := FALSE;
	RETURN;
END_IF

// Rezerwacja struktury danych dla zapytania
IF NOT bReturnDataBusy OR bReturnDataReserved_SelMachParams THEN
	IF NOT bCmdSended THEN	// Przygotowanie danych do zapytania
		stSqlComandData.nCmdState:= nSQL_CmdExecState.New;
		stSqlComandData.nCmdType:=nSQL_CmdTypes.SelMachineParams;
		stSqlComandData.byExecutingNodeNb:=0;
	(*	stSqlComandData.bWaitForDataReturn:=TRUE;
		IF diParamsId <> 0 THEN		// Rodzaj zapytania zależy od tego po czym chcemy wyszukiwać zestawy parametrów 
			stSqlComandData.sCmdExpression :=  'SELECT ParamsData, CRC_Sum, ParamsSizeInBytes FROM [dbo].[ProductionMachineParameters] WHERE Id = {IdLineStation}';
			stSqlComandData.stCmdData.IdLineStation := diParamsId;
		ELSE
			stSqlComandData.sCmdExpression :=  'SELECT ParamsData, CRC_Sum, ParamsSizeInBytes FROM [dbo].[ProductionMachineParameters] WHERE Active = 1 AND MachineNumber = {MachineNumber} AND IdLineStation = {IdLineStation} AND IdComposedPart = {IdComposedPart}';
			stSqlComandData.stCmdData.MachineNumber := iMachineNumber;
			stSqlComandData.stCmdData.IdLineStation := stRetDataLineStation.IdStacji;
			stSqlComandData.stCmdData.IdComposedPart := stRetDataLineStation.IdOutComposedPart;
		END_IF	*)
		stSqlComandData.pReturnedData := ADR(stRetDataMachParams);
		stSqlComandData.uiReturnedDataSize := SIZEOF(stRetDataMachParams);
		stSqlComandData.bSQL_OK := stSqlComandData.bSQL_Done := FALSE;
		// Próba dodania komendy do kolejki
		IF I_SqlCore <> 0 AND_THEN  I_SqlCore.mAddCmdToQueue(ADR(stSqlComandData)) THEN
			bCmdSended := bReturnDataBusy := bReturnDataReserved_SelMachParams := TRUE;		// Zajęcie struktury danych
			MEMSET(destAddr := ADR(stRetDataMachParams), n := SIZEOF(stRetDataMachParams), fillByte:= 0);		// Czyszczenie danych 
		ELSE
			bResultOk := FALSE;
			m_SqlSelMachineParamsData := bCmdAddError := TRUE;
		END_IF
	ELSIF stSqlComandData.bSQL_Done THEN	// Przetwarzanie zapytania SQL zakończone 
		IF stSqlComandData.bSQL_OK THEN
			IF stRetDataMachParams.DataSize = UINT_TO_INT(uiParamsDataSize) THEN	// Rozmiar parametrów zgodny
				IF INT_TO_WORD(stRetDataMachParams.CRC16sum) = F_DATA_TO_CRC16_CCITT(pData := ADR(stRetDataMachParams.StructRawData), cbData := INT_TO_UDINT(stRetDataMachParams.DataSize), crc:= 0) THEN
					MEMCPY(srcAddr := ADR(stRetDataMachParams.StructRawData), destAddr := pParamsData, n:= uiParamsDataSize);
					bParametersUpdated := TRUE;
				ELSE		// Niezgodne sumy CRC - raczej niemożliwe
					mNewEvent(nInputErrorID := nPIM_ErrorCodes.ParamsMismatchPLCandDB, nEventType := nPIM_EventClasses.Alarm, tMessageTime := T#0S);
					MEMCPY(srcAddr := ADR(stRetDataMachParams.StructRawData), destAddr := pParamsData, n:= uiParamsDataSize);
				END_IF
			ELSE
				mNewEvent(nInputErrorID := nPIM_ErrorCodes.ParamsMismatchPLCandDB, nEventType := nPIM_EventClasses.Alarm, tMessageTime := T#0S);
				MEMSET(destAddr := pParamsData, n := uiParamsDataSize, fillByte:= 0);		// Czyszczenie danych parametrów
				MEMCPY(srcAddr := ADR(stRetDataMachParams.StructRawData), destAddr := pParamsData, n:= MIN(uiParamsDataSize,INT_TO_UINT(stRetDataMachParams.DataSize)));
			END_IF
		ELSE	// Jeśli nie zwrócono żadnego rekordu brak pasujących parametrów - trzeba najpierw przesłać parametry do DB
			mNewEvent(nInputErrorID := nPIM_ErrorCodes.NoMatchingParamsForComponent, nEventType := nPIM_EventClasses.Alarm, tMessageTime := T#0S);
			bNoMatchingParams := TRUE;	;
		END_IF
		bSelMachineParamsData := TRUE;	// Odświeżenie parametrów w strukturze PIM, skasowanie zmiennej bCmdSended
		bResultOK := stSqlComandData.bSQL_OK;
		m_SqlSelMachineParamsData := bUpdateData := TRUE;
	END_IF
END_IF
pParamsData := ADR(stRetDataMachParams.StructRawData);
bProcessing := bCmdSended AND NOT stSqlComandData.bSQL_Done;
END_METHOD

ACTION ACT_PimCmdsHandling:
// TImer gotowości PIMu (komunikacja itp jest OK)
fbTOF_PimWorking(IN:= FALSE, PT:= T#5M, Q=> bPIM_Working);		// TImer o gotowości systemu PIM

//Obsługa komunikatów z PIMu
IF stPimInOut.sCmdPIM2PLC <> '' AND NOT bCmdReaded THEN
	stPimInOut.sCmdPIM2PLC := F_ToLCase(stPimInOut.sCmdPIM2PLC);
	sStringToParse := F_ToLCase(stPimInOut.sCmdPIM2PLC);
	WHILE sStringToParse <> '' DO
		sActCmd := fPIM_GetCmdPar(sParseString := sStringToParse);
		IF sActCmd = 'lifebit' THEN
			fbTOF_PimWorking(IN:= TRUE);
		ELSIF sActCmd = 'rework' THEN
			IF fPIM_GetCmdPar(sParseString := sStringToParse) = 'true' THEN
				nReworkMenuStatus := nPIM_ReworkSelect.yes;
				iCtr_PIM_PartsNOK := LIMIT(0,iCtr_PIM_PartsNOK - 1,32767);
			ELSE
				nReworkMenuStatus := nPIM_ReworkSelect.no;
			END_IF
		ELSIF sActCmd = 'sendmachineparamstodb' THEN			// Zapisuje w bazie danych parametry pracy dla aktualnego złożenia jako aktywne 
			bMachParamsSendToDB:= TRUE;
		ELSIF sActCmd = 'readmachineparamsfromdb' THEN
			bMachParamsReadFromDB := TRUE;	// Wymuszenie pobrania parametrów z bazy danych
			bMachineParamsOK := FALSE;		// Zatrzymanie pracy na czas pobrania elementów
		ELSIF sActCmd = 'retool' THEN		// Pobiera z bazy danych parametry dla danego złożenia
			bRetool := TRUE;	// Wymuszenie pobrania parametrów z bazy danych
			bMachineParamsOK := FALSE;		// Zatrzymanie pracy na czas pobrania elementów
		ELSIF sActCmd = 'newboxout' THEN
			iOutBoxQty:= STRING_TO_INT(fPIM_GetCmdPar(sParseString := sStringToParse));
			iOutBoxTargetQty:= STRING_TO_INT(fPIM_GetCmdPar(sParseString := sStringToParse));
		ELSIF sActCmd = 'nokreported' THEN	// Zgłoszenie po wykonaniu operacji - do ustalenia źródło zgłoszenia
			sActCmd := fPIM_GetCmdPar(sParseString := sStringToParse);				
			IF sActCmd = 'fprevstation' THEN
				nReoprtedNokSource:= nPIM_ReportedNokSource.FromPrevStation;
			ELSIF sActCmd = 'fmach' THEN
				nReoprtedNokSource:= nPIM_ReportedNokSource.FromMach;				
			ELSIF sActCmd = 'fbox' THEN
				nReoprtedNokSource:= nPIM_ReportedNokSource.FromBox;
			ELSE
				nReoprtedNokSource:= nPIM_ReportedNokSource.Error_UnknownSource;			
			END_IF
		ELSIF sActCmd = 'logged' THEN
			sUserRole:= fPIM_GetCmdPar(sParseString := sStringToParse);
			sUserLang:= fPIM_GetCmdPar(sParseString := sStringToParse);
		ELSIF sActCmd = '' THEN
			MEMMOVE(srcAddr := ADR(asUnsuportedCmds[1]), destAddr := ADR(asUnsuportedCmds[2]), n := 4*SIZEOF(asUnsuportedCmds[1]));
			asUnsuportedCmds[1] := 'EmptyString';
		ELSE
			MEMMOVE(srcAddr := ADR(asUnsuportedCmds[1]), destAddr := ADR(asUnsuportedCmds[2]), n := 4*SIZEOF(asUnsuportedCmds[1]));
			asUnsuportedCmds[1] := sActCmd;
		END_IF
	END_WHILE
	bCmdReaded := TRUE;
ELSE
	stPimInOut.sCmdPIM2PLC := '';
	bCmdReaded := FALSE;
	nReoprtedNokSource:= nPIM_ReportedNokSource.none;
	nReworkMenuStatus := nPIM_ReworkSelect.none;
END_IF


//Obsługa komunikatów z PIMu
fbTON_CmdPLC2PIM_Reset(IN:= stPimInOut.sCmdPLC2PIM <> '', PT:= T#100MS);
IF fbTON_CmdPLC2PIM_Reset.Q THEN
	stPimInOut.sCmdPLC2PIM := '';
	bCmdPlc2PimSended := FALSE;
END_IF
bCmdPlc2PimSended R= stPimInOut.sCmdPLC2PIM = '';



(*	Komendy do wysłania:
	- Wyloguj użytkownika?
	- Zgłoś usterkę maszyny
*)
END_ACTION

ACTION ACT_SqlDataReturnCmd:

bSQLCmdError := FALSE;
fbTON_CmdHangedUp(IN:= bReturnDataBusy AND NOT stSqlComandData.bSQL_Done, PT:= T#10S);
IF fbTON_CmdHangedUp.Q THEN
	fbTON_CmdHangedUp(IN:= FALSE);
	stSqlComandData.bSQL_Done := TRUE;
	stSqlComandData.bSQL_OK := FALSE;
	fbLogger.mAppendCurrentLine(bBreakLine := TRUE, sAddSep := '', sAppendText:= 'Sql command Hungedup, service reset');
	uiCtr_CmdReset:= uiCtr_CmdReset +1; 
END_IF


// Jeśli chcemy serwisowo sprawdzić działanie funkcji ustawić zmienne wejściowe w odpowiedni sposób oraz ustawić zmienną w If np. bSelectStationId
IF bSelectStationId THEN
	IF NOT bUpdateData THEN
		m_SqlSelLineStationId(bProcessing => bPimCmdProcessing);
	END_IF
	IF stSqlComandData.bSQL_Done THEN
		IF stSqlComandData.bSQL_OK THEN		// Pobranie danych OK
		//	stRetDataLineStation.AutoControlMachineParams := FALSE;
			stStationStatus.stStationSqlData := stRetDataLineStation; 
			bStationIdValid := TRUE;
		ELSE 
			bSQLCmdError := TRUE;
		END_IF
		bCmdSended := bSelectStationId := FALSE;
		bReturnDataBusy := bReturnDataReserved_StationId := FALSE;
	//	MEMSET(destAddr := ADR(stDBCmdData), n := SIZEOF(stDBCmdData), fillByte:= 0);		// Czyszczenie danych zapytania
	ELSE
		IF NOT bPimCmdProcessing THEN
			bSQLCmdError := TRUE;
			bCmdSended := bSelectStationId := FALSE;
			bReturnDataBusy := bReturnDataReserved_StationId := FALSE;		
		END_IF
	END_IF
END_IF

IF bInsertStatus THEN 
	IF NOT bUpdateData THEN
		m_SqlSelInsStatus(bStatus:=bLastStatus , sErrCode:= sLastErrCode, bSustein := FALSE, bProcessing => bPimCmdProcessing);
	END_IF
	IF stSqlComandData.bSQL_Done THEN	
		IF stSqlComandData.bSQL_OK THEN
			bStatusSavedOK := TRUE;
			iCtr_StatusSaveOK := iCtr_StatusSaveOK + 1; 
			mSendCmdToPIM(sCmd := CONCAT(STR1:='StatusId:', STR2:= LINT_TO_STRING(liLPartStatusId)));
			IF bLockAfterStatusSave THEN
				IF stPimInOut.sErrorCodePLC = '' THEN
					iConvTMP := nPIM_ErrorCodes.UnKnownLock;
					stPimInOut.sErrorCodePLC := INT_TO_STRING(iConvTMP);
				END_IF
				stPimInOut.bAlarmPLC :=  stPimInOut.bNonBlockingAlarm := FALSE;
				stPimInOut.bWorkBlock_PLC := TRUE;				
			END_IF
		ELSE
			bSQLCmdError := TRUE;
			iCtr_StatusSaveError := iCtr_StatusSaveError + 1; 
			mSendCmdToPIM(sCmd := 'StatusSaveError');
			IF bLockAfterStatusSave THEN
				IF stPimInOut.sErrorCodePLC = '' THEN
					iConvTMP := nPIM_ErrorCodes.UnKnownLock;
					stPimInOut.sErrorCodePLC := INT_TO_STRING(iConvTMP);
				END_IF
				stPimInOut.bWorkBlock_PLC := TRUE;
			END_IF
		END_IF
		bLockAfterStatusSave :=	bCmdSended := bInsertStatus := FALSE;		
		bReturnDataBusy := bReturnDataReserved_InsOperStat := FALSE;
	//	MEMSET(destAddr := ADR(stDBCmdData), n := SIZEOF(stDBCmdData), fillByte:= 0);		// Czyszczenie danych zapytania
	ELSE
		IF NOT bPimCmdProcessing THEN
			bSQLCmdError := TRUE;
			bCmdSended := bInsertStatus := FALSE;
			bReturnDataBusy := bReturnDataReserved_InsOperStat := FALSE;		
		END_IF
	END_IF
END_IF


IF bSelPreviousStatus THEN 
	IF NOT bUpdateData THEN
		m_SqlSelLastOperationStatus(sCodeDM:= sLastDMCode, bProcessing => bPimCmdProcessing);
	END_IF
	IF stSqlComandData.bSQL_Done THEN
		IF  stSqlComandData.bSQL_OK THEN
			bPreviousOperationStatus := bPreviousOperationStatus;		
		ELSE
			bSQLCmdError := TRUE;
		END_IF
		bCmdSended := bSelPreviousStatus := FALSE;
		bReturnDataBusy := bReturnDataReserved_SelLastOperStat := FALSE;
	ELSE
		IF NOT bPimCmdProcessing THEN
			bSQLCmdError := TRUE;
			bCmdSended := bSelPreviousStatus := FALSE;
			bReturnDataBusy := bReturnDataReserved_SelLastOperStat := FALSE;		
		END_IF
	END_IF	
END_IF

IF bSelMachineParamsData THEN
	IF NOT bUpdateData THEN
		m_SqlSelMachineParamsData(diParamsId := 0, pParamsData:= 0, uiParamsDataSize := 0, bProcessing => bPimCmdProcessing);
	END_IF
	IF stSqlComandData.bSQL_Done THEN
		bSQLCmdError := NOT stSqlComandData.bSQL_OK;		
		bCmdSended := bSelMachineParamsData := FALSE;
		bReturnDataBusy := bReturnDataReserved_SelMachParams := FALSE;
	ELSE
		IF NOT bPimCmdProcessing THEN
			bSQLCmdError := TRUE;
			bCmdSended := bSelMachineParamsData := FALSE;
			bReturnDataBusy := bReturnDataReserved_SelMachParams := FALSE;		
		END_IF
	END_IF
END_IF

IF bSelMachineParamsCRC THEN
	IF NOT bUpdateData THEN
		m_SqlSelMachineParamsCRC(liIdCompossedPart := 0, bProcessing => bPimCmdProcessing);
	END_IF
	IF stSqlComandData.bSQL_Done THEN
		IF stSqlComandData.bSQL_OK THEN
			diMachineParamsInsertId := diMachineParamsInsertId;
		ELSE
			bSQLCmdError := TRUE;
		END_IF
		bCmdSended := bSelMachineParamsCRC := FALSE;
		bReturnDataBusy := bReturnDataReserved_SelMachParamsCRC := FALSE;
	ELSE 
		IF NOT bPimCmdProcessing THEN 
			bSQLCmdError := TRUE;
			bCmdSended := bSelMachineParamsCRC := FALSE;
			bReturnDataBusy := bReturnDataReserved_SelMachParamsCRC := FALSE;		
		END_IF
	END_IF
END_IF

IF bInsMachineParamsData THEN
	IF NOT bUpdateData THEN
		m_SqlInsMachineParamsData(pParamsData := 0, uiParamsDataSize := 0, wCrcSumOfParameters := 0, bProcessing => bPimCmdProcessing);
	END_IF
	IF stSqlComandData.bSQL_Done THEN
		IF stSqlComandData.bSQL_OK THEN
			diMachineParamsInsertId := diMachineParamsInsertId;
		ELSE
			bSQLCmdError := TRUE;
		END_IF
		bCmdSended := bInsMachineParamsData := FALSE;
		bReturnDataBusy := bReturnDataReserved_InsMachParams := FALSE;
	ELSE 
		IF NOT bPimCmdProcessing THEN 
			bSQLCmdError := TRUE;
			bCmdSended := bInsMachineParamsData := FALSE;
			bReturnDataBusy := bReturnDataReserved_InsMachParams := FALSE;		
		END_IF
	END_IF
END_IF

ACT_UpdatePimOutput();
bUpdateData := FALSE;
END_ACTION

ACTION ACT_UpdatePimOutput:
//stPimInOut := stPimInternal;		// Aktualizacja danych wyjściowych wewnętrzną strukturą
END_ACTION

METHOD FB_init : BOOL
VAR_INPUT
	bInitRetains : BOOL; // if TRUE, the retain variables are initialized (warm start / cold start)
	bInCopyCode : BOOL;  // if TRUE, the instance afterwards gets moved into the copy code (online change)
	I_Sql:I_SQL_Core;
END_VAR
I_SqlCore := I_Sql;
END_METHOD

// Metoda zwraca strukturę do zapytania SQL uzupełnioną o dane z bloczka stanowiska
METHOD mGetStationData : stPIM_StationStatus
VAR_OUTPUT
	sCMD				: STRING;		// Zdarzenie jednostkowe/ rozkaz z PIMu np uaktualniono dane itp.
	bUserLogged			: BOOL;			// Użytkownik zalogowany
	bPIM_Active			: BOOL;			// Info o aktywności systemu PIM
	bTestMode			: BOOL;			// Aktywny tryb testowy
	bWorkPermittion		: BOOL;			// Informacja o zezwoleniu na pracę sumarycznie
	bWorkBlockPIM		: BOOL;			// Informacja o zezwoleniu na pracę z PIM
	bWorkBlockPLC		: BOOL;			// Informacja o zezwoleniu na pracę z PLC
	bConfirmation		: BOOL;			// Informacja o potwierdzeniu błędu
	bExternalMessage	: BOOL;			// Informacja o aktywnym komunikacie zewnętrznym
	nExtErrorClass		: nPIM_EventClasses;			// Informacja o aktywnym błędzie zewnętrznym
	bEventWaitInQueue	: BOOL;			// Info, że zdarzenie zewnętrzne czeka w kolejce
	nMachState			: nPIM_MachineStates;	// Aktualny status maszyny
	bOperInProgress		: BOOL;			// TRUE gdy operacja trwa
	bOperEnded			: BOOL;			// Impuls gdy operacja zakończona
	bOperStatus			: BOOL;			// Status ostatniej operacji
	nReworkSelected 	: nPIM_ReworkSelect;	// Operator wybrał Opcje reworku na tak lub nie
	nReoprtedNok 		: nPIM_ReportedNokSource;	// Operator zgłosił NOKa
END_VAR
mGetStationData:= stStationStatus;

sCMD := sCmdToSendToMachine;
sCmdToSendToMachine := '';
bUserLogged := fbTON_UserLogedDeleyed.Q;
bPIM_Active := stPimInOut.bPIMActive;
bWorkPermittion	:= bWorkPermitt;	
bConfirmation := stPimInOut.bConfirmEvent;
bTestMode := stPimInOut.bTestMode;
nExtErrorClass := nActEventClass;
nMachState := nMachineState;

bOperInProgress := nMachineState = nPIM_MachineStates._4_OperationInProgress ;
bOperEnded := bOperationEnded OR nMachineState = nPIM_MachineStates._5_OperationEndedOK ;
bOperStatus := bLastStatus;
nReworkSelected:= nReworkMenuStatus;
nReoprtedNok := nReoprtedNokSource;
END_METHOD

METHOD INTERNAL mNewEvent : BOOL
VAR_INPUT
	nInputErrorID:	INT;	// Kod błędu w postaci inta (do przekonwertowania)
	nEventType: nPIM_EventClasses;	// ROdzaj nowego zdarzenia
	tMessageTime: TIME:= T#3S;		// Czas na wyświetlenie wiadomości- ma znaczenie tylko dla wiadomości (po tym czasie lub po starcie nowej operacji wiadomość znika)
END_VAR
VAR
	sType: STRING;
	iConvTMP: INT;
END_VAR
IF nInputErrorID <> 0 THEN		// Kod błędu podany przez Enum
	stPimInOut.sErrorCodePLC := INT_TO_STRING(nInputErrorID);
ELSE	// Brak kodu błędu -
	iConvTMP := nPIM_ErrorCodes.UnKnownLock;
	stPimInOut.sErrorCodePLC := INT_TO_STRING(iConvTMP);
END_IF		

CASE nEventType OF 
	nPIM_EventClasses.Error:		// Błąd związany z częścią - trzeba bezwzględnie zapisać status i wtedy wystawić odpowiednie bity
		m_SqlSelInsStatus(bStatus := FALSE, sErrCode := stPimInOut.sErrorCodePLC, bSustein := TRUE);
		bStatusSaveTriggered := bInsertStatus := TRUE;
		bLockAfterStatusSave := TRUE;	
		iCtr_Errors:= iCtr_Errors + 1; 
		
	nPIM_EventClasses.Alarm:
		stPimInOut.bAlarmPLC := NOT stPimInOut.bWorkBlock_PLC;	// Jeśli jest już aktywne blokowanie, nie aktywuj alarmu tylko zmień kod błędu
		stPimInOut.bNonBlockingAlarm := FALSE;
		m_SqlInsAdditionalError(sErrCode:= stPimInOut.sErrorCodePLC);
		
	nPIM_EventClasses.AlarmAutoConfirm:
		stPimInOut.bNonBlockingAlarm := stPimInOut.bAlarmPLC := NOT stPimInOut.bWorkBlock_PLC;
		m_SqlInsAdditionalError(sErrCode:= stPimInOut.sErrorCodePLC);
		
	nPIM_EventClasses.Message:
		stPimInOut.bNonBlockingAlarm := stPimInOut.bAlarmPLC := NOT stPimInOut.bWorkBlock_PLC;
		fbTON_MessageTimer(IN:= TRUE, PT := tMessageTime);
END_CASE	
nActEventClass := nEventType;
ACT_UpdatePimOutput();

nEventType := nEventType;
nErrorID := nInputErrorID;
sType := TO_STRING(nEventType);
fbFormatStr(sFormat := 'Nowy event typ- %s, Id- %d',arg1 := F_STRINGEx(sType), arg2 := F_INT(nErrorID));  
fbLogger.mAddLine(sTextToSave := fbFormatStr.sOut );
iWorkStep := 99;
END_METHOD

METHOD INTERNAL mSendCmdToPIM : BOOL
VAR_INPUT
	sCmd: STRING;
END_VAR
IF stPimInOut.sCmdPLC2PIM = '' THEN		// Cmd Empty
	stPimInOut.sCmdPLC2PIM := CONCAT(STR1:= sCmd, STR2:= ';');
ELSE	// Not empty - check if cmd isnt sended
	IF NOT bCmdPlc2PimSended THEN
		IF RIGHT(STR:= stPimInOut.sCmdPLC2PIM, SIZE:= 1) <> ';' THEN		// Separator are not present
			stPimInOut.sCmdPLC2PIM := CONCAT(STR1:= stPimInOut.sCmdPLC2PIM, STR2:= ';');	
		END_IF
		stPimInOut.sCmdPLC2PIM := CONCAT(STR1:= sCmd, STR2:= 'sCmd');
		stPimInOut.sCmdPLC2PIM := CONCAT(STR1:= stPimInOut.sCmdPLC2PIM, STR2:= ';');
	ELSE		// Write cmd in bufer		
		IF sCmdPlc2PimBufer = '' THEN		// Cmd Empty
			sCmdPlc2PimBufer := CONCAT(STR1:= sCmd, STR2:= ';');
		ELSE	// Not empty
			IF RIGHT(STR:= sCmdPlc2PimBufer, SIZE:= 1) <> ';' THEN		// Separator are not present
				sCmdPlc2PimBufer := CONCAT(STR1:= sCmdPlc2PimBufer, STR2:= ';');	
			END_IF
			sCmdPlc2PimBufer := CONCAT(STR1:= sCmd, STR2:= 'sCmd');
			sCmdPlc2PimBufer := CONCAT(STR1:= sCmdPlc2PimBufer, STR2:= ';');
		END_IF
	END_IF
END_IF
mSendCmdToPIM := TRUE;
END_METHOD

END_FUNCTION_BLOCK

// SQL/I_SQL_Core
INTERFACE I_SQL_Core

METHOD IsCoreWork : BOOL
VAR_INPUT
END_VAR
END_METHOD

METHOD mAddCmdToQueue : BOOL
VAR_INPUT
	pNewCmdData:POINTER TO stSQL_ClientNode;
END_VAR
VAR_OUTPUT
	nErrorID:nSQL_ErrorCodes;
END_VAR
END_METHOD

END_INTERFACE

// PIM/POUs/fPIM_GetCmdPar
FUNCTION fPIM_GetCmdPar : STRING
VAR_IN_OUT
	sParseString:STRING(255);
END_VAR
VAR_OUTPUT
	bEnd:BOOL;	// Koniec komendy
	bPar:BOOL;	// Parametr do wczytania
END_VAR
VAR
	i:INT;
	sActChar: STRING(1);
	iStrLen: INT;
END_VAR

// Komendy postaci „Cmd[:Par1][:Par2][:Par3];" - pierwszy element to komenda, parametry są po dwukropku, komendę zakańcza średnik
// Funkcja wczytuje ciąg znaków aż do znaku : , ; lub końca stringu oraz zwraca wczytaną treść bez znaku separatora lub końca
iStrLen := LEN(STR := sParseString); 
sParseString := F_ToLCase(sParseString);
IF iStrLen > 0 THEN	// Jeśli string wejściowy pusty zakończ przetwarzanie.
	FOR i := 1 TO iStrLen BY 1 DO
		sActChar := MID(STR:= sParseString, LEN := 1 , POS := i);	// Sprawdzenie znaku na pozycji i
		IF sActChar = ';' OR sActChar = ':' THEN	// Jeśli aktualny indeks to koniec komendy/parametru to podziel string w tym mijescu i zwróć dane	
			fPIM_GetCmdPar := LEFT (STR := sParseString, SIZE := i-1);		// Komenda
			sParseString := RIGHT(STR := sParseString, SIZE := iStrLen - i);	// Pozostały string do sprawdzenia
			IF sActChar = ':' THEN
				bPar := TRUE;
			ELSE
				bEnd := TRUE;
			END_IF
			EXIT;	
		ELSIF i = iStrLen THEN		
			fPIM_GetCmdPar := sParseString;
			sParseString := '';
			EXIT;	
		END_IF
	END_FOR
END_IF

END_FUNCTION

// PIM/POUs/fbPIM_Station_V3
FUNCTION_BLOCK FINAL fbPIM_Station_V3 IMPLEMENTS  I_PIM, I_SqlCmds

VAR_INPUT
	stPimInOut: REFERENCE TO stPIM_ServiceInOuts;	// Dane pobierane z/ wysyłane do systemu PIM
	sLineName : STRING(31);							// Nazwa linii w systemie PIM
	sStationName : STRING(31);						// Nazwa stanowiska w systemie PIM
	iMachineNumber : INT:= 1;						// Numer maszyny na stanowisku
	bIsHidden : BOOL:= FALSE;						// Czy ukrywanie zapisu statusu (jeśli TRUE część nie jest liczona jako wyjściowa ze stanowiska)
	sPrevStationName : STRING(31);					// Do sprawdzenia statusu ostatniej operacji - jeśli funkcja nieużywana zostaw puste
	stStationSettings:stPIM_StationSettings;		// Ustawienia stanowiska	
END_VAR
VAR_OUTPUT
	bStationDataOK: BOOL;
	bUserLogged: BOOL;							// Użytkownik zalogowany
	bTestMode: BOOL;
	bWorkPermitt: BOOL;
	nErrorID:nPIM_ErrorCodes;
	bOperationEnded: BOOL;
	bOperationStatus: BOOL;
	stStationStatus: stPIM_StationStatus;
	nReoprtedNokSource: nPIM_ReportedNokSource;
	nReworkMenuStatus:nPIM_ReworkSelect;
END_VAR
VAR
	nActIntErrorClass, nActExtErrorClass: nPIM_EventClasses;	// Informacje o aktualnym typie alarmu
	I_Machine: I_StationMachine;				// Interfejs do obsługi maszyn - pobranie danych z maszyny (głównie parametry pracy)
	I_SqlCore:	I_SQL_Core;						// Interfejs do obsługi zapytań SQL
	bPIM_Working:BOOL;							// Informacja o działaniu systemu PIM (Odświeżany Cykliczny lifeBit)
	nMachineState: nPIM_MachineStates;
	iWorkStep :INT;
	stSqlComandData:stSQL_ClientNode;			// Struktura do zapytań z danymi powrotnymi (struktura jest blokowana na czas zapytania)
	stSqlComandDataTMP:stSQL_ClientNode;		// Struktura do zapytań bez danych powrotnych (podczas tworzenia zapytania dynamicznie tworzona kopia)
	bSelectStationId, bInsertStatus, bSelPreviousStatus, bSelMachineParamsData, bInsMachineParamsData, bSelMachineParamsCRC: BOOL;
	bReturnDataBusy: BOOL;
	liLPartStatusId: LINT;
	
	stRetDataLineStation	: stSQL_RetDataProdLineStat;	
	stRetDataMachParams		: stSQL_RetDataProdMachParams;	
	stRetDataUserRole		: stSQL_RetDataUserRole;
	iConvTMP:INT;
	bCmdAddError: BOOL;
	bCmdSended: BOOL;
	bPimCmdProcessing: BOOL:= FALSE;
	sActCmd: STRING;
	fbTOF_PimWorking: TOF;
	asUnsuportedCmds:ARRAY [1..5] OF STRING;
	bReturnDataReserved_StationId, bReturnDataReserved_InsOperStat, bReturnDataReserved_SelLastOperStat,
		bReturnDataReserved_SelMachParams, bReturnDataReserved_InsMachParams, bReturnDataReserved_SelMachParamsCRC: BOOL;		// Zmienne rezerwujące strukturę danych dla zapytań które zwracają dane z DB
	diMachineParamsInsertId: DINT;
	bUpdateData: BOOL;
	fbTON_ConfirmReset: TON;
	wCrcSumInDb:WORD;
	bMachineParamsOK: BOOL;
	bMachParSql_Processing: BOOL;
	bMachParSql_Result_OK: BOOL;
	diLastParamsInsID: DINT;
	sStringToParse: STRING(255);
	bCmdReaded:BOOL;
	
	sUserRole: STRING;
	sUserLang: STRING(3);
	fbTON_MessageTimer, fbTON_ServiceMessageTimer:TON;	// TImer wyświetlania alarmu lub wiadomości w dolnym pasku
		
	bLockAfterStatusSave: BOOL;
	
	bNewOperationInProgress: BOOL;		// Inforamcja o rozpoczętej operacji, kasowana po zakończeniu operacji i zapisie statusu operacji
	bStatusSaveTriggered: BOOL;		// Flaga o wystawieniu zapisu statusu do DB
	bStatusSavedOK: BOOL;				// Informacja o poprawnym zapisie statusu
	bPreviousOperationStatus: BOOL;
	
	wCrcSumInMachine: WORD;
	bStationDataOK_TemporaryAlowed: BOOL;
	iPartsQtyPermittTemporary: INT;
	bParReadBusy: BOOL;
	pParametersPtr: POINTER TO BYTE;
	uiParametersSize: UINT;
	bMachParamsSendToDB, bMachParamsReadFromDB: BOOL;	// Zapis/odczyt parametrów pracy maszyny do/z bazy danych

	
	// Kolejka alarmów
	iNextEventCodeEnum:	INT;				// Kod następnego błędu w kolejce 
	nNextEeventType: nPIM_EventClasses;			// Rozdzaj następnego błędu w kolejce
	tNextEeventMessageTime: TIME:= T#3S;		// Czas wyświetlania następnej wiadomości w kolejce 
	bNextEventSource:BOOL;						// Źródło następnego błędu w kolejce 0-Int, 1-Ext

	bParamsInMachineUpdated: BOOL;
	bRetool: BOOL;
	iOutBoxQty,	iOutBoxTargetQty: INT;
	bRefreshData: BOOL;
	sCmdToSendToMachine: STRING;
	fbTON_AutoReset: TON;
	iMemPimWorkStep: INT;
	aiPimWorkStepHistoric: ARRAY [1..10] OF INT;
	fbLogger:fbTextDataLogger;
	sFormat:STRING(2047);
	fbFormatStr2:FB_FormatString2;
	fbFormatStr:FB_FormatString;
	iCtr_Operations, iCtr_OperationsInterrupted, iCtr_OperationsEndedOK, iCtr_OperEndedOK_Method, iCtr_OperationsEndedNOK: INT;
	iCtr_PIM_PartsOK, iCtr_PIM_PartsNOK, iCtr_PIM_ReworkYes, iCtr_PIM_PartOK_SaveError, iCtr_PIM_PartNOK_SaveError, iCtr_StatusSaveOK, iCtr_StatusSaveError, iCtr_Errors: INT;
	iCtrMem_Operations, iCtrMem_OperationsInterrupted, iCtrMem_OperationsEndedOK, iCtrMem_OperEndedOK_Method, iCtrMem_OperationsEndedNOK: INT;
	iCtrMem_PIM_PartsOK, iCtrMem_PIM_PartsNOK, iCtrMem_PIM_ReworkYes, iCtrMem_PIM_PartOK_SaveError, iCtrMem_PIM_PartNOK_SaveError, iCtrMem_StatusSaveOK, iCtrMem_StatusSaveError, iCtrMem_Errors: INT;
	
	iCtr_NewEventCalls, iCtr_NewEventCalls_ER, iCtr_NewEventCalls_AL, iCtr_NewEventCalls_Other,
			iCtr_NewIntEventCalls, iCtr_NewComEventCalls_ER, iCtr_NewComEventCalls_AL, iCtr_NewComEventCalls_Other: INT;
	iCtrMem_NewEventCalls, iCtrMem_NewEventCalls_ER, iCtrMem_NewEventCalls_AL, iCtrMem_NewEventCalls_Other, 
			iCtrMem_NewIntEventCalls, iCtrMem_NewComEventCalls_ER, iCtrMem_NewComEventCalls_AL, iCtrMem_NewComEventCalls_Other: INT;
	bWriteHistoricData: BOOL;
	bTestZapisu: BOOL;
	fbTON_UserLogedDeleyed: TON;
	fbTON_CmdHangedUp: TON;
	bLastStatus: BOOL;
	sLastErrCode: STRING(10);

	bNewOperationStartedMethod,	bNewOperationEndedOKMethod, bOperationEndedErrorMethod: BOOL;	// Informacjeo wywołaniu bloczka z metod

	sLastDMCode: STRING(255);
	bTestAdditionalErrorSave: BOOL;
	bTestResult: BOOL;
	bTestComprAirCtrSave: BOOL;
	bTestEnergyCtrSave: BOOL;
	fbTON_BlindAlarm: TON;
	uiCtr_CmdReset: UINT;
	liRetoolParamsIdFromPIM: LINT;
	fbTON_StepTimeout:TON;
	fbTON_CmdPLC2PIM_Reset: TON;
	bCmdPlc2PimSended: BOOL;
	sCmdPlc2PimBufer: STRING(255);
	bSaveDefectRelation: BOOL;
	bTestDefectRealtionSave: BOOL;
	sStationAlias: STRING(31);
	bUserLoggedMem: BOOL;
	fbTON_WriteErrorCode2Status: TON;
END_VAR
VAR PERSISTENT
	liIdOutCompossedPartMemory:LINT;			// Id ostatniego elementu składanego na stanowisku z zatwierdzonymi parametrami
	wLastParametersCrcMemory: WORD;			// Suma CRC ostatnich zgodnych parametrów
END_VAR


//	Wychwycenie znaczników pewnych zdarzeń
fbTON_UserLogedDeleyed(IN:= stPimInOut.bUserLogged, PT:= T#100MS, Q=> bUserLogged);
fbLogger(sNetId := '', sPreambule := GVL_Aircom.stAC_DT_Data.sLogTimeString,);
bRefreshData S= stPimInOut.bUserLogged AND NOT bUserLoggedMem;
bTestMode := stPimInOut.bTestMode;

IF NOT stPimInOut.bUserLogged AND bUserLoggedMem THEN
	stPimInOut.sStatusNokAndErrorID := '';
END_IF
bUserLoggedMem := stPimInOut.bUserLogged;

// Zapisanie relacji do błędu
fbTON_WriteErrorCode2Status(PT:=T#100MS);
IF fbTON_WriteErrorCode2Status.Q THEN
	fbTON_WriteErrorCode2Status.IN:= FALSE;
	stPimInOut.sStatusNokAndErrorID := CONCAT(STR1:= LINT_TO_STRING(liLPartStatusId), STR2:= CONCAT(STR1:= ':',STR2:= stPimInOut.sErrorCodePLC));
END_IF

// W przypadku braku aktywnego błędu oraz obecnego błędu w kolejce dodaj błąd z kolejki
IF iNextEventCodeEnum <> 0 AND (nActIntErrorClass = nPIM_EventClasses.NoError AND nActextErrorClass = nPIM_EventClasses.NoError) THEN
	IF bNextEventSource THEN
		mNewEvent(iEventId := iNextEventCodeEnum, nEventType := nNextEeventType, tMessageTime := tNextEeventMessageTime);
	ELSE 
		mNewlnternalEvent(nInputErrorID := nErrorID, nEventType := nNextEeventType, tMessageTime := tNextEeventMessageTime);
	END_IF
	iNextEventCodeEnum := 0;	// Kasowanie alarmu w kolejce
END_IF


fbTON_BlindAlarm(IN:= NOT fbTON_BlindAlarm.Q AND stPimInOut.bConfirmEvent AND (nActIntErrorClass = nPIM_EventClasses.NoError AND nActextErrorClass = nPIM_EventClasses.NoError), PT:= T#200MS);
IF fbTON_BlindAlarm.Q THEN		// Zabezpieczenie - brak aktywnego alarmu w PLC a przyszło potwierdzenie
	mNewlnternalEvent(nInputErrorID := nPIM_ErrorCodes.UnKnownAlarm, nEventType := nPIM_EventClasses.Alarm, tMessageTime := T#0S);			
ELSIF (nActExtErrorClass >= nPIM_EventClasses.AlarmAutoConfirm OR nActIntErrorClass >= nPIM_EventClasses.AlarmAutoConfirm) AND NOT stPimInOut.bAlarmPLC AND NOT stPimInOut.bWorkBlock_PLC THEN
	stPimInOut.bNonBlockingAlarm := nActExtErrorClass = nPIM_EventClasses.AlarmAutoConfirm OR nActIntErrorClass = nPIM_EventClasses.AlarmAutoConfirm;
	stPimInOut.bAlarmPLC := TRUE;
ELSIF (nActExtErrorClass = nPIM_EventClasses.Error OR nActIntErrorClass = nPIM_EventClasses.Error) AND NOT stPimInOut.bWorkBlock_PLC AND NOT bLockAfterStatusSave THEN
	stPimInOut.bWorkBlock_PLC := TRUE;
END_IF

bOperationStatus := bLastStatus;


(*IF NOT stPimInternal.bPIMActive AND NOT (iWorkStep <> -1) THEN
	iWorkStep := -1;
	stPimInternal.sWiadomoscPLC := 'PIM_NotActive';
	fbTON_ServiceMessageTimer.IN:= FALSE;
	fbTON_AutoReset(IN:= nMachineState = nPIM_MachineStates._8_WaitForReset , PT:= T#5S);
END_IF*)

IF iMemPimWorkStep <> iWorkStep THEN
	MEMMOVE(srcAddr := ADR(aiPimWorkStepHistoric[1]), destAddr := ADR(aiPimWorkStepHistoric[2]), n:= 9*SIZEOF(aiPimWorkStepHistoric[1]));
	aiPimWorkStepHistoric[1]:= iMemPimWorkStep;
END_IF
iMemPimWorkStep:=iWorkStep;

bOperationEnded:= FALSE;

bWorkPermitt := stPimInOut.bTestMode OR NOT stPimInOut.bPIMActive OR 
					(bUserLogged AND NOT stPimInOut.bWorkBlock_PIM AND NOT stPimInOut.bWorkBlock_PLC
					AND (NOT stPimInOut.bAlarmPLC OR stPimInOut.bNonBlockingAlarm)
					AND bMachineParamsOK AND bStationDataOK AND NOT bRetool AND NOT bMachParamsReadFromDB AND NOT bMachParamsSendToDB) AND (nActIntErrorClass <> nPIM_EventClasses.Error AND nActIntErrorClass <> nPIM_EventClasses.Alarm);
				
CASE iWorkStep OF
	
	0:		// Inicjalizacja stanowiska
		fbLogger.sDirectoryToSave:= CONCAT(STR1:= GVL_Aircom.sLogsPath, STR2:=CONCAT(STR1:='PIM\', STR2:= sStationName));
		fbFormatStr(sFormat := 'W%d_PIMlog_%s_m%d.txt',
			arg1 := F_WORD(GVL_Aircom.stAC_DT_Data.wWeekNb), 
			arg2 := F_STRINGEx(sStationName), 
			arg3 := F_INT(iMachineNumber), sOut => fbLogger.sFileNameWithFormat );  
		sStationAlias := prStationAlias;// CONCAT(STR1:= CONCAT(STR1:= sStationName, '_'), INT_TO_STRING(iMachineNumber));
			
		stStationStatus.sLine := sLineName;
		stStationStatus.sStation := sStationName;
		stStationStatus.sNazwaStanowiska:= CONCAT(STR1:= CONCAT(STR1:= sStationName, '_'), INT_TO_STRING(iMachineNumber));
		stStationStatus.iMachineNumber := iMachineNumber;
		stStationStatus.bIsHidden := bIsHidden;
		stSqlComandData.sStation := stSqlComandDataTMP.sStation := stStationStatus.sNazwaStanowiska;
		bMachineParamsOK := bStationDataOK := bStationDataOK_TemporaryAlowed := FALSE;
		bSelectStationId := TRUE;	// Pobranie danych stanowiska z bazy danych
		fbTON_StepTimeout(IN:= FALSE);
		iWorkStep := 1;
		
	1:	// Pobranie parametrów pracy maszyny 
		fbTON_StepTimeout(IN:= TRUE, PT:= T#10S);
		IF I_Machine <> 0 THEN
			IF I_Machine.mGetParamsData(bTestParams := FALSE, bBusy => bParReadBusy, pMachineParametersStruct => pParametersPtr, uiMachineParametersSize => uiParametersSize, wActualCRC16SumInMachine => wCrcSumInMachine) THEN
				iWorkStep := 5;
			ELSIF NOT bParReadBusy THEN
				mNewlnternalEvent(nInputErrorID := nPIM_ErrorCodes.MachineParametersNoUpdated, nEventType := nPIM_EventClasses.Alarm, tMessageTime := T#0S);
			END_IF
		ELSE	// Nie podłączony interfejs brak komunikacji z maszyną
			{warning <'Zmienić na konkretny rodzaj błędu'>}
			mNewlnternalEvent(nInputErrorID := nPIM_ErrorCodes.ProgramError, nEventType := nPIM_EventClasses.Alarm, tMessageTime := T#0S);
		END_IF
		IF iWorkStep <> 1 THEN 	fbTON_StepTimeout(IN:= FALSE);	END_IF
		
	5:	// Oczekiwanie na Pobranie danch stacji z bazy danych 
		fbTON_StepTimeout(IN:= TRUE, PT:= T#10S );
		IF NOT bSelectStationId THEN
			IF stRetDataLineStation.IdStacji <> 0 THEN	
				bStationDataOK := TRUE;
				iWorkStep := 6;
			ELSE
				mNewlnternalEvent(nInputErrorID := nPIM_ErrorCodes.SelectStationIdError, nEventType := nPIM_EventClasses.Alarm, tMessageTime := T#0S);
			END_IF
		ELSIF fbTON_StepTimeout.Q THEN
			mNewlnternalEvent(nInputErrorID := nPIM_ErrorCodes.SelectStationIdError, nEventType := nPIM_EventClasses.Alarm, tMessageTime := T#0S);
		END_IF
		IF iWorkStep <> 5 THEN 	fbTON_StepTimeout(IN:= FALSE);	END_IF
	
	6:	// Sprawdzenie czy w DB jest zdefiniowane złożenie wyjściowe, czy są parametry dla złożenia oraz czy pasują do danych w PLC 
		fbTON_StepTimeout(IN:= TRUE, PT:= T#10S );
		IF stStationSettings.bCheckMachineSettings THEN
			IF stRetDataLineStation.IdOutComposedPart <> 0 THEN
				IF bMachParamsReadFromDB THEN
					bMachParamsSendToDB := FALSE;
					iWorkStep := 50;
				ELSIF bMachParamsSendToDB THEN
					iWorkStep := 60;
				ELSIF stRetDataLineStation.CrcSumOfParams <> 0 THEN
					IF wCrcSumInMachine = stRetDataLineStation.CrcSumOfParams THEN		// Parametry są zgodne
						bMachineParamsOK := TRUE;
						liIdOutCompossedPartMemory := stRetDataLineStation.IdOutComposedPart;
						wLastParametersCrcMemory := stRetDataLineStation.CrcSumOfParams;
						iWorkStep := 10;
					ELSE	// Parametry niezgodne
						mNewlnternalEvent(nInputErrorID := nPIM_ErrorCodes.ParamsMismatchPLCandDB, nEventType := nPIM_EventClasses.Alarm, tMessageTime := T#0S);
					END_IF
				ELSE
					mNewlnternalEvent(nInputErrorID := nPIM_ErrorCodes.NoMatchingParamsForComponent, nEventType := nPIM_EventClasses.Alarm, tMessageTime := T#0S);
				END_IF
			ELSE
				mNewlnternalEvent(nInputErrorID := nPIM_ErrorCodes.NoConfiguredOutPart, nEventType := nPIM_EventClasses.Alarm, tMessageTime := T#0S);
			END_IF	
		ELSE
			bMachineParamsOK := TRUE;
			iWorkStep := 10;	
		END_IF
		IF iWorkStep <> 6 THEN 	fbTON_StepTimeout(IN:= FALSE);	END_IF

	10:	// Inicjalizacja zakończona OK, oczekiwanie na operacje z maszyny
		bRetool := bMachParamsReadFromDB := bMachParamsSendToDB := FALSE;
		IF bRefreshData THEN	// Odświeżenie danych stanowiska
 			iWorkStep := 0;
			bRefreshData := FALSE;			
		ELSIF bRetool OR bMachParamsReadFromDB THEN
			bMachParamsSendToDB := FALSE;
			iWorkStep := 50;
		ELSIF bMachParamsSendToDB THEN
			iWorkStep := 60;
		ELSIF nMachineState = nPIM_MachineStates._3_NewOperationStarted OR bNewOperationStartedMethod THEN
			fbLogger.mAppendCurrentLine(bBreakLine := FALSE, sAddSep := '', sAppendText:= 'NewOpStarted');
			IF bStationDataOK_TemporaryAlowed THEN		// Jeśli parametry dopuszczone warunkowo co 100 sztuk zablokuj stanowisko
				iPartsQtyPermittTemporary := iPartsQtyPermittTemporary;
				IF iPartsQtyPermittTemporary > 100 THEN
					bStationDataOK_TemporaryAlowed := FALSE; 
					iPartsQtyPermittTemporary := 0;
				END_IF
			END_IF
			iCtr_Operations:= iCtr_Operations +1;
			bStatusSaveTriggered := bStatusSavedOK := FALSE;
			iWorkStep := 15;
		END_IF
		bNewOperationStartedMethod := FALSE;
		
	15:	// Operacja trwa, oczekiwanie na zakończenie (możliwy pomiar czasu cyklu)
		IF nMachineState = nPIM_MachineStates._2_ReadyForNewOperation THEN
			iCtr_Operations:= iCtr_Operations -1;
			iCtr_OperationsInterrupted:= iCtr_OperationsInterrupted +1; 
			fbLogger.mAppendCurrentLine(bBreakLine := FALSE, sAddSep := '', sAppendText:= ', OperInterrupted');
			iWorkStep := 10;
		ELSIF nMachineState = nPIM_MachineStates._5_OperationEndedOK THEN
			iCtr_OperationsEndedOK:= iCtr_OperationsEndedOK +1;
			bOperationEnded:= TRUE;
			IF bStatusSaveTriggered THEN
				fbLogger.mAppendCurrentLine(bBreakLine := FALSE, sAddSep := '', sAppendText:= ', OperEndedOK_StatusSaveInProgress');
				iWorkStep := 20;
			ELSE
				fbLogger.mAppendCurrentLine(bBreakLine := FALSE, sAddSep := '', sAppendText:= ', OperEndedOK_StatusSaveNotTrigered');
				mNewlnternalEvent(nInputErrorID := nPIM_ErrorCodes.ProgramError, nEventType := nPIM_EventClasses.Alarm, tMessageTime := T#0S);
			END_IF
		ELSIF nMachineState = nPIM_MachineStates._7_ErrorOccurr THEN
			iCtr_OperationsEndedNOK:= iCtr_OperationsEndedNOK +1;
			bOperationEnded:= TRUE;
			IF nActExtErrorClass = nPIM_EventClasses.Error AND NOT bStatusSaveTriggered THEN
				fbLogger.mAppendCurrentLine(bBreakLine := FALSE, sAddSep := '', sAppendText:= ', OperEndedNOK_StatSavNotTriged');
				mNewlnternalEvent(nInputErrorID := nPIM_ErrorCodes.ProgramError, nEventType := nPIM_EventClasses.Error, tMessageTime := T#0S);
			ELSIF bStatusSaveTriggered THEN
				fbLogger.mAppendCurrentLine(bBreakLine := FALSE, sAddSep := '', sAppendText:= ', OperEndedNOK_NoStatusSave');
				iWorkStep := 20;
			ELSE
				iWorkStep := 25;
			END_IF
		END_IF
		
	20:	// Oczekiwanie na zapis statusu - sprawdzenie wyniku
		IF stStationSettings.bSkipCheckStatusSaveResult THEN
			fbLogger.mAppendCurrentLine(bBreakLine := FALSE, sAddSep := '', sAppendText:= ', CSSR_Skiped');	
			iWorkStep := 25;			
		ELSIF NOT bInsertStatus THEN
			IF bStatusSavedOK THEN
				fbLogger.mAppendCurrentLine(bBreakLine := FALSE, sAddSep := '', sAppendText:= ', StatusSaved');
				iWorkStep := 25;	
			ELSE
				fbLogger.mAppendCurrentLine(bBreakLine := FALSE, sAddSep := '', sAppendText:= ', StatusNotSaved');
				mNewlnternalEvent(nInputErrorID := nPIM_ErrorCodes.StatusSaveError, nEventType := nPIM_EventClasses.Alarm, tMessageTime := T#0S);
			END_IF
		END_IF
		
	25:	// Oczekiwanie na zakończenie operacji
		IF nMachineState = nPIM_MachineStates._2_ReadyForNewOperation THEN 
			fbLogger.mAppendCurrentLine(bBreakLine := TRUE, sAddSep := '', sAppendText:= ', OperEnded_BaseState_2');
			bNewOperationInProgress := FALSE;
			iWorkStep := 10;	
		END_IF
		
	50:	// Odczyt parametrów z bazy danych - pobranie aktualnych parametrów z bazy danych i maszyny
		IF I_Machine.mGetParamsData(bTestParams := FALSE, bBusy => bParReadBusy, pMachineParametersStruct => pParametersPtr, uiMachineParametersSize => uiParametersSize, wActualCRC16SumInMachine => wCrcSumInMachine) THEN
			bParamsInMachineUpdated := FALSE;
			iWorkStep := 52;
		ELSIF NOT bParReadBusy THEN
			mNewlnternalEvent(nInputErrorID := nPIM_ErrorCodes.ParamsReadFromDB_Error, nEventType := nPIM_EventClasses.Alarm, tMessageTime := T#0S);
		END_IF
		
	52:	//
		IF uiParametersSize < 1000 THEN
			IF m_SqlSelMachineParamsData(diParamsId := 0, pParamsData := pParametersPtr , uiParamsDataSize := uiParametersSize, bProcessing=> bMachParSql_Processing, bResultOK=> bMachParSql_Result_OK, bParametersUpdated => bParamsInMachineUpdated) THEN
				IF bMachParSql_Result_OK AND bParamsInMachineUpdated THEN
					iWorkStep := 54;
				ELSE 
					mNewlnternalEvent(nInputErrorID := nPIM_ErrorCodes.ParamsReadFromDB_Error, nEventType := nPIM_EventClasses.Alarm, tMessageTime := T#0S);
				END_IF
			ELSIF NOT bMachParSql_Processing THEN		// Błąd SQL
				mNewlnternalEvent(nInputErrorID := nPIM_ErrorCodes.ParamsReadFromDB_Error, nEventType := nPIM_EventClasses.Alarm, tMessageTime := T#0S);
			END_IF
		END_IF	
		
	54:	// Odczyt parametrów z bazy danych - Dane odczytane poprawnie
		 bRetool := bMachParamsReadFromDB := FALSE;
		iWorkStep := 0;
		
	60:	// Zapis parametrów do bazy danych - pobranie aktualnych parametrów z bazy danych i maszyny
		IF I_Machine.mGetParamsData(bTestParams := FALSE, bBusy => bParReadBusy, pMachineParametersStruct => pParametersPtr, uiMachineParametersSize => uiParametersSize, wActualCRC16SumInMachine => wCrcSumInMachine) THEN
			iWorkStep := 62;
		ELSIF NOT bParReadBusy THEN
			mNewlnternalEvent(nInputErrorID := nPIM_ErrorCodes.ParamsSaveToDB_Error, nEventType := nPIM_EventClasses.Alarm, tMessageTime := T#0S);
		END_IF
		
	62:	// Zapis parametrów do bazy danych - wysłanie pobranych parametrów do bazy danych
		IF m_SqlInsMachineParamsData(pParamsData := pParametersPtr, uiParamsDataSize := uiParametersSize, wCrcSumOfParameters := wCrcSumInMachine, bProcessing=> bMachParSql_Processing, bResultOK=> bMachParSql_Result_OK, diParamsId => diLastParamsInsID) THEN
			IF bMachParSql_Result_OK THEN		// Parametry pobrane,
				iWorkStep := 64;
			ELSE 
				mNewlnternalEvent(nInputErrorID := nPIM_ErrorCodes.ParamsSaveToDB_Error, nEventType := nPIM_EventClasses.Alarm, tMessageTime := T#0S);
			END_IF
		ELSIF NOT bMachParSql_Processing THEN		// Błąd SQL
			mNewlnternalEvent(nInputErrorID := nPIM_ErrorCodes.ParamsSaveToDB_Error, nEventType := nPIM_EventClasses.Alarm, tMessageTime := T#0S);
		END_IF
			
	64:	// Zapis parametrów do bazy danych - Parametry zapisane poprawnie
	//	stPimTMP.sCmdPLC2PIM := CONCAT(STR1:= CONCAT(STR1:='ParamsSaved:', STR2:= DINT_TO_STRING(diLastParamsInsID)), STR2:= ';');	Opcjonalne potwierdzenie zapisu do PIMu
		bMachParamsSendToDB := FALSE;
		iWorkStep := 0;
		
	99:
		IF (stPimInOut.bConfirmEvent OR (nErrorID = nPIM_ErrorCodes.SelectStationIdError AND fbTON_AutoReset.Q ))
			 AND nActIntErrorClass <> nPIM_EventClasses.NoError THEN
			
			fbLogger.mAddLine(sTextToSave := CONCAT(STR1:= 'Reset bledu - wewnetrznego', STR2:= stPimInOut.sErrorCodePLC ) );
			IF 	nErrorID = nPIM_ErrorCodes.MachineParametersNoUpdated		// Błąd w inicjalizacji stanowiska do pracy
					OR nErrorID = nPIM_ErrorCodes.SelectStationIdError 
					OR nErrorID = nPIM_ErrorCodes.NoConfiguredOutPart
					OR nErrorID = nPIM_ErrorCodes.NoMatchingParamsForComponent
					OR nErrorID = nPIM_ErrorCodes.ParamsMismatchPLCandDB THEN
				iWorkStep := 0;
				
			ELSIF nErrorID = nPIM_ErrorCodes.StatusSaveError THEN			// Gdy błąd zapisu statusu spróbuj jeszcze raz
				m_SqlSelInsStatus(bStatus := bLastStatus, sErrCode := sLastErrCode, bSustein := TRUE);
				iWorkStep := 20;
			ELSIF nErrorID = nPIM_ErrorCodes.ParamsReadFromDB_Error			// Gdy błąd odczytu parametrów z bazy danych spróbuj jeszcze raz
				  OR nErrorID = nPIM_ErrorCodes.ParamsMismatchPLCandDB
				  OR nErrorID = nPIM_ErrorCodes.NoMatchingParamsForComponent  THEN		
				IF bMachParamsSendToDB THEN			// Jeśli błąd w pobraniu, a aktywny również zapis parametrów najpierw zapisz parametry, potem pobierz
					iWorkStep := 60;
				ELSE
					iWorkStep := 50;
				END_IF
				
			ELSIF nErrorID = nPIM_ErrorCodes.ParamsSaveToDB_Error THEN		// Gdy błąd zapisu parametrów w bazie danych spróbuj jeszcze raz
				iWorkStep := 60;
			ELSE
				iWorkStep := 0;
			END_IF
			nErrorID := nPIM_ErrorCodes.NoError;
			stPimInOut.bNonBlockingAlarm := stPimInOut.bAlarmPLC := stPimInOut.bWorkBlock_PLC := FALSE;
			stPimInOut.sErrorCodePLC := '';
			nActIntErrorClass := nPIM_EventClasses.NoError;
			stPimInOut.bConfirmEvent := FALSE;
		ELSIF nActIntErrorClass = nPIM_EventClasses.Message THEN
				iWorkStep := 10;
		ELSE
			IF nActIntErrorClass = nPIM_EventClasses.NoError AND nActExtErrorClass = nPIM_EventClasses.NoError 
					AND (NOT stPimInOut.bAlarmPLC AND NOT stPimInOut.bWorkBlock_PLC) AND NOT bLockAfterStatusSave THEN
				mNewlnternalEvent(nInputErrorID := nPIM_ErrorCodes.UnKnownAlarm, nEventType := nPIM_EventClasses.Error, tMessageTime := T#0S);	
			END_IF
		END_IF
	
END_CASE
fbTON_AutoReset(IN:= iWorkStep = 99 AND NOT fbTON_AutoReset.Q, PT:= T#10S);

ACT_PimCmdsHandling();		// Obsługa komend z/do PIMu
ACT_SqlDataReturnCmd();		// Obsługa zapytań SQL do DB


// Automatyczne kasowanie aktualnej wiadomości po zadanym czasie wyświetlania lub alarmu przy starcie nowej operacji
fbTON_MessageTimer();
IF stPimInOut.bNonBlockingAlarm AND (fbTON_MessageTimer.Q OR nMachineState = nPIM_MachineStates._3_NewOperationStarted) THEN
	fbTON_MessageTimer(IN:= FALSE);
	stPimInOut.sErrorCodePLC := '';
	stPimInOut.bNonBlockingAlarm := stPimInOut.bAlarmPLC := FALSE;
	IF nActIntErrorClass = nPIM_EventClasses.Message OR nActIntErrorClass = nPIM_EventClasses.AlarmAutoConfirm THEN
		nActIntErrorClass := nPIM_EventClasses.Message;
	 END_IF
	 IF nActExtErrorClass = nPIM_EventClasses.Message OR nActExtErrorClass = nPIM_EventClasses.AlarmAutoConfirm THEN
		nActExtErrorClass := nPIM_EventClasses.Message;
	 END_IF
END_IF

fbTON_ServiceMessageTimer();		// Reset wiadomości serwisowej
IF fbTON_ServiceMessageTimer.Q THEN
	fbTON_ServiceMessageTimer(IN:= FALSE);
	stPimInOut.sPlcServiceMessage := '';
END_IF



	
		
IF GVL_Aircom.stAC_DT_Data.bNew_Shift OR bTestZapisu THEN
	fbFormatStr(sFormat := 'W%d_PIMlog_%s_m%d.txt',
		arg1 := F_WORD(GVL_Aircom.stAC_DT_Data.wWeekNb), 
		arg2 := F_STRINGEx(sStationName), 
		arg3 := F_INT(iMachineNumber), sOut => fbLogger.sFileNameWithFormat ); 
	iCtrMem_Operations := iCtr_Operations;
	iCtrMem_OperationsInterrupted := iCtr_OperationsInterrupted;
	iCtrMem_OperationsEndedOK := iCtr_OperationsEndedOK;
	iCtrMem_OperEndedOK_Method := iCtr_OperEndedOK_Method;
	iCtrMem_OperationsEndedNOK := iCtr_OperationsEndedNOK;
	iCtrMem_PIM_PartsOK := iCtr_PIM_PartsOK;
	iCtrMem_PIM_PartsNOK := iCtr_PIM_PartsNOK;
	iCtrMem_PIM_ReworkYes := iCtr_PIM_ReworkYes;
	iCtrMem_PIM_PartOK_SaveError := iCtr_PIM_PartOK_SaveError;
	iCtrMem_PIM_PartNOK_SaveError := iCtr_PIM_PartNOK_SaveError;
	iCtrMem_StatusSaveOK := iCtr_StatusSaveOK;
	iCtrMem_StatusSaveError := iCtr_StatusSaveError;
	iCtrMem_Errors := iCtr_Errors;
	iCtrMem_NewEventCalls:= iCtr_NewEventCalls;
	iCtrMem_NewIntEventCalls:= iCtr_NewIntEventCalls;
	iCtrMem_NewEventCalls_ER := iCtr_NewEventCalls_ER;
	iCtrMem_NewEventCalls_AL := iCtr_NewEventCalls_AL;
	iCtrMem_NewEventCalls_Other := iCtr_NewEventCalls_ER;
	iCtrMem_NewIntEventCalls:= iCtr_NewIntEventCalls; 
	iCtrMem_NewComEventCalls_ER:= iCtr_NewComEventCalls_ER; 
	iCtrMem_NewComEventCalls_AL:= iCtr_NewComEventCalls_AL;
	iCtrMem_NewComEventCalls_Other:= iCtr_NewComEventCalls_Other;
	iCtr_Operations:= iCtr_OperationsInterrupted:= iCtr_OperationsEndedOK:= iCtr_OperEndedOK_Method:= iCtr_OperationsEndedNOK:= 0; 
	iCtr_PIM_PartsOK:= iCtr_PIM_PartsNOK:= iCtr_PIM_ReworkYes:= iCtr_PIM_PartOK_SaveError := iCtr_PIM_PartNOK_SaveError:= iCtr_StatusSaveOK:= iCtr_StatusSaveError:= iCtr_Errors:= 0;
	iCtr_NewEventCalls:= iCtr_NewEventCalls_ER:= iCtr_NewEventCalls_AL:= iCtr_NewEventCalls_Other:= iCtr_NewIntEventCalls:= 0;
	iCtr_NewComEventCalls_ER:= iCtr_NewComEventCalls_AL:= iCtr_NewComEventCalls_Other:= 0;
	fbLogger.mAddLine(sTextToSave := CONCAT(STR1:= 'Nowa zmiana - ', STR2:= UINT_TO_STRING( GVL_Aircom.stAC_DT_Data.uiShiftNumber) ));
	fbLogger.mSaveBuffor();
	bTestZapisu := FALSE;
	bWriteHistoricData := TRUE;
END_IF
IF bWriteHistoricData AND fbLogger.bBufferEmpty THEN
	fbFormatStr(sFormat := 'PrevShiftReport: Oper-%d, OperInt-%d, OperOK-%d, OperOK_M-%d, OperNOK-%d',
		arg1 := F_INT(iCtrMem_Operations), 
		arg2 := F_INT(iCtrMem_OperationsInterrupted), 
		arg3 := F_INT(iCtrMem_OperationsEndedOK), 
		arg4 := F_INT(iCtrMem_OperEndedOK_Method), 
		arg5 := F_INT(iCtrMem_OperationsEndedNOK));  
	fbLogger.mAddLine(sTextToSave := fbFormatStr.sOut );
	fbFormatStr(sFormat := 'PrevShiftReport: PartsPIM_OK-%d, PartsPIM_NOK-%d, PartsPIM_ReworkYes-%d, PartsPIM_OK_missed-%d, PartsPIM_NOK_Missed-%d',
		arg1 := F_INT(iCtrMem_PIM_PartsOK), 
		arg2 := F_INT(iCtrMem_PIM_PartsNOK), 
		arg4 := F_INT(iCtrMem_PIM_ReworkYes),
		arg5 := F_INT(iCtrMem_PIM_PartOK_SaveError), 
		arg6 := F_INT(iCtrMem_PIM_PartNOK_SaveError));  
	fbLogger.mAddLine(sTextToSave := fbFormatStr.sOut );
	fbFormatStr(sFormat := 'PrevShiftReport: StatusSaveOK-%d, StatusSaveError-%d, Errors-%d, CmdReset- %d',
		arg1 := F_INT(iCtrMem_StatusSaveOK), 
		arg2 := F_INT(iCtrMem_StatusSaveError), 
		arg3 := F_INT(iCtrMem_Errors), 
		arg4 := F_UINT(in:=uiCtr_CmdReset));  
	uiCtr_CmdReset := 0;
	fbLogger.mAddLine(sTextToSave := fbFormatStr.sOut );	
	fbLogger.mSaveBuffor();
	bWriteHistoricData := FALSE;
END_IF

fbTON_ConfirmReset(IN:= stPimInOut.bConfirmEvent, PT:= T#500MS);
stPimInOut.bConfirmEvent R= fbTON_ConfirmReset.Q;

ACT_UpdatePimOutput();		// Aktualizacja danych wyjściowych wewnętrzną strukturą

PROPERTY PartsCtr_NOK : INT
GET
PartsCtr_NOK := iCtr_PIM_PartsNOK;
END_GET
END_PROPERTY

PROPERTY PartsCtr_OK : INT
GET
PartsCtr_OK := iCtr_PIM_PartsOK;
END_GET
END_PROPERTY

// The number of actually displayed error code ex "601"
PROPERTY prActiveErrorCode : STRING
GET
prActiveErrorCode := stPimInOut.sErrorCodePLC;
END_GET
END_PROPERTY

(* Get CMD Value from PIM*)
PROPERTY prCMD : STRING
GET
IF __ISVALIDREF(stPimInOut) THEN
	prCMD := sCmdToSendToMachine;
	sCmdToSendToMachine := '';	
END_IF
END_GET
END_PROPERTY

(* Get info *)
PROPERTY prCurrentMachineState : nPIM_MachineStates
GET
prCurrentMachineState := nMachineState;
END_GET
END_PROPERTY

(* Get info *)
PROPERTY prErrorClassExt : nPIM_EventClasses
GET
prErrorClassExt := nActExtErrorClass;
END_GET
END_PROPERTY

(* Get info *)
PROPERTY prErrorConfirmActive : BOOL
GET
IF __ISVALIDREF(stPimInOut) THEN
	prErrorConfirmActive := stPimInOut.bConfirmEvent;
END_IF
END_GET
END_PROPERTY

(* Get info *)
PROPERTY prExternalEvtWaitInQueue : BOOL
GET
prExternalEvtWaitInQueue := iNextEventCodeEnum <> 0 AND bNextEventSource;
END_GET
END_PROPERTY

(* Get info is PIM is active*)
PROPERTY prLastSavedStatus : BOOL
GET
prLastSavedStatus := bLastStatus;
END_GET
END_PROPERTY

(* Get info is PIM is active*)
PROPERTY prNokReportedSource : nPIM_ReportedNokSource
GET
prNokReportedSource := nReoprtedNokSource;
END_GET
END_PROPERTY

(* Get info is PIM is active*)
PROPERTY prOperEnded : BOOL
GET
prOperEnded := nMachineState = nPIM_MachineStates._5_OperationEndedOK OR nMachineState = nPIM_MachineStates._7_ErrorOccurr;
END_GET
END_PROPERTY

(* Get info is PIM is active*)
PROPERTY prOperInProgress : BOOL
GET
prOperInProgress := nMachineState >= nPIM_MachineStates._3_NewOperationStarted AND nMachineState <= nPIM_MachineStates._6_ReturningToBaseState;
END_GET
END_PROPERTY

(* Get info is PIM is active*)
PROPERTY prPimActive : BOOL
GET
IF __ISVALIDREF(stPimInOut) THEN
	prPimActive := stPimInOut.bPIMActive;
END_IF
END_GET
END_PROPERTY

(* Get info *)
PROPERTY prPimBlockWork : BOOL
GET
IF __ISVALIDREF(stPimInOut) THEN
	prPimBlockWork := stPimInOut.bWorkBlock_PIM;
END_IF
END_GET
END_PROPERTY

(* Get info *)
PROPERTY prPlcBlockWork : BOOL
GET
IF __ISVALIDREF(stPimInOut) THEN
	prPlcBlockWork := stPimInOut.bWorkBlock_PLC;
END_IF
END_GET
END_PROPERTY

(* Get info is PIM is active*)
PROPERTY prReworkStatus : nPIM_ReworkSelect
GET
prReworkStatus := nReworkMenuStatus;
END_GET
END_PROPERTY

// Get info if station data is correctlly downloaded from database
PROPERTY prStationDataOK : BOOL
GET
prStationDataOK := bStationDataOK;
END_GET
END_PROPERTY

(* Get info is test mode is active*)
PROPERTY prTestMode : BOOL
GET
IF __ISVALIDREF(stPimInOut) THEN
	prTestMode := stPimInOut.bTestMode;
END_IF
END_GET
END_PROPERTY

(* Get info is user are logged?*)
PROPERTY prUserLogged : BOOL
GET
IF __ISVALIDREF(stPimInOut) THEN
	prUserLogged := stPimInOut.bUSerLogged;
END_IF
END_GET
END_PROPERTY

(* Get info *)
PROPERTY prWorkPermission : BOOL
GET
IF __ISVALIDREF(stPimInOut) THEN
	prWorkPermission := stPimInOut.bTestMode OR NOT stPimInOut.bPIMActive OR (stPimInOut.bUSerLogged AND NOT stPimInOut.bWorkBlock_PIM AND NOT stPimInOut.bWorkBlock_PLC
					AND (NOT stPimInOut.bAlarmPLC OR stPimInOut.bNonBlockingAlarm) AND bStationDataOK AND NOT bRetool AND NOT bMachParamsReadFromDB 
					AND NOT bMachParamsSendToDB) AND (nActIntErrorClass <> nPIM_EventClasses.Error AND nActIntErrorClass <> nPIM_EventClasses.Alarm);
ELSE
	prWorkPermission := FALSE;
END_IF
END_GET
END_PROPERTY

(* Get info is that machine is EOL*)
PROPERTY prIsEol : BOOL
GET
prIsEol := stRetDataLineStation.IsEOL;
END_GET
END_PROPERTY

(* Get Station name followed by machine number ex: 'CA01PL19_1'*)
PROPERTY prPartCodeNumber : STRING(250)
GET
prPartCodeNumber := stRetDataLineStation.PartCodeNumber;
END_GET
END_PROPERTY

(* Get Hidden status info*)
PROPERTY prIsHidden : BOOL
GET
prIsHidden := bIsHidden;
END_GET
END_PROPERTY

(* Get Line name ex: 'CA01PL'*)
PROPERTY prLineName : STRING(31)
GET
prLineName := sLineName;
END_GET
END_PROPERTY

(* Get Machine number*)
PROPERTY prMachNumber : INT
GET
prMachNumber := iMachineNumber;
END_GET
END_PROPERTY

(* Get Station name followed by machine number ex: 'CA01PL19_1'*)
PROPERTY prStationAlias : STRING(31)
GET
prStationAlias := CONCAT(STR1:= CONCAT(STR1:= sStationName, '_'), INT_TO_STRING(iMachineNumber));
END_GET
END_PROPERTY

(* Get Station name ex: 'CA01PL19'*)
PROPERTY prStationName : STRING(31)
GET
prStationName := sStationName;
END_GET
END_PROPERTY

// Zapis do DB dodatkowego kodu błędu - jeśli rozkaz dodany do kolejki zmienna wyjściowa ma wartość TRUE, jeśli nie (błąd dodania) FALSE
METHOD m_SqlInsAdditionalError : BOOL
VAR_INPUT
	sErrCode:STRING(10);		// Kod błędu do wysłania
END_VAR
VAR
	bResult:BOOL;
END_VAR
IF sErrCode <> '' AND stRetDataLineStation.IdStacji <> 0 THEN
	stSqlComandDataTMP.nCmdState:= nSQL_CmdExecState.New;
	stSqlComandDataTMP.nCmdType:=nSQL_CmdTypes.InsAdditionalError;
	stSqlComandDataTMP.bWaitForDataReturn:=FALSE;
	sFormat := 'INSERT INTO [dbo].[ProductionLineStationAdditionalError] (IdLineStation, MachineNumber, IdMachineError) VALUES (%d, %d, COALESCE( (SELECT Id FROM [dbo].[ProductionMachineError] WHERE Active = 1 AND Code = $'%s$'), -9223372036854775285))';
	fbFormatStr2(pFormatString := ADR(sFormat),
			arg1:= F_DINT(stRetDataLineStation.IdStacji),
			arg2:= F_INT(iMachineNumber),
			arg3:= F_STRINGEx(sErrCode),
			pDstString := ADR(stSqlComandDataTMP.sCmdExpression), nDstSize := SIZEOF(stSqlComandDataTMP.sCmdExpression));

	stSqlComandDataTMP.pReturnedData := 0;
	stSqlComandDataTMP.uiReturnedDataSize := 0;	
	IF I_SqlCore <> 0 THEN
		bResult := I_SqlCore.mAddCmdToQueue(ADR(stSqlComandDataTMP));
	END_IF
	m_SqlInsAdditionalError := bResult;
ELSE
	m_SqlInsAdditionalError := FALSE;
END_IF
END_METHOD

// Zapis do DB licznika zużycia powietrza - jeśli rozkaz dodany do kolejki zwraca TRUE, jeśli nie FALSE
METHOD m_SqlInsCompressedAirConsumption : BOOL
VAR_INPUT
	rActCompressedAirConsumption:REAL;		// Wartość licznika zużycia sprężonego powietrza
END_VAR
IF rActCompressedAirConsumption <> 0 AND stRetDataLineStation.IdLinii <> 0 THEN
	stSqlComandDataTMP.nCmdState:= nSQL_CmdExecState.New;
	stSqlComandDataTMP.nCmdType:=nSQL_CmdTypes.InsCompressedAirCons;
	stSqlComandDataTMP.bWaitForDataReturn:=FALSE;
	
	sFormat := 'INSERT INTO `ProductionConsumption_CompressedAir` (`IdLine`, `CounterValue`, `ValueUnit`) VALUES ( %d, %.3f, $'m3$')';
	fbFormatStr2(pFormatString := ADR(sFormat),
			arg1:= F_DINT(stRetDataLineStation.IdLinii),
			arg2:= F_REAL(rActCompressedAirConsumption),
			pDstString := ADR(stSqlComandDataTMP.sCmdExpression), nDstSize := SIZEOF(stSqlComandDataTMP.sCmdExpression));
	stSqlComandDataTMP.pReturnedData := 0;
	stSqlComandDataTMP.uiReturnedDataSize := 0;	
	IF I_SqlCore <> 0 THEN
		m_SqlInsCompressedAirConsumption := I_SqlCore.mAddCmdToQueue(ADR(stSqlComandDataTMP));
	END_IF	
ELSE
	m_SqlInsCompressedAirConsumption := FALSE;
END_IF
END_METHOD

// Zapis do DB relacji ostatniego statusu z kodem błędu - jeśli rozkaz dodany do kolejki zwraca TRUE, jeśli nie FALSE
METHOD m_SqlInsDefectRelation : BOOL
VAR_INPUT
	sErrCode:STRING(10);			// Kod błędu
END_VAR
IF sErrCode <> '' THEN
	stSqlComandDataTMP.nCmdState:= nSQL_CmdExecState.New;
	stSqlComandDataTMP.nCmdType:=nSQL_CmdTypes.InsDefectRelation;
	stSqlComandDataTMP.bWaitForDataReturn:=FALSE;
	
	sFormat := 'INSERT INTO [dbo].[ProductionMachinePartsStatusDefectRelation] (IdPartStatus, IdMachineError) values (%d, (SELECT Id FROM [dbo].[ProductionMachineError] WHERE Active = 1 AND Code = $'%s$'))';
	fbFormatStr2(pFormatString := ADR(sFormat),
			arg1:= F_LINT(liLPartStatusId),
			arg2:= F_STRINGEx(sErrCode),
			pDstString := ADR(stSqlComandDataTMP.sCmdExpression), nDstSize := SIZEOF(stSqlComandDataTMP.sCmdExpression));
	stSqlComandDataTMP.pReturnedData := 0;
	stSqlComandDataTMP.uiReturnedDataSize := 0;	
	IF I_SqlCore <> 0 THEN
		m_SqlInsDefectRelation := I_SqlCore.mAddCmdToQueue(ADR(stSqlComandDataTMP));
	END_IF
ELSE
	m_SqlInsDefectRelation := FALSE;
END_IF
END_METHOD

// Zapis do DB licznika zużycia energi na stanowisku - jeśli rozkaz dodany do kolejki zwraca TRUE, jeśli nie FALSE
METHOD m_SqlInsEnergyConsumption : BOOL
VAR_INPUT
	rActEnergyConsumption:REAL;			// Wartość licznika zużycia energii elektrycznej
END_VAR
IF rActEnergyConsumption <> 0 AND stRetDataLineStation.IdStacji <> 0 THEN
	stSqlComandDataTMP.nCmdState:= nSQL_CmdExecState.New;
	stSqlComandDataTMP.nCmdType:=nSQL_CmdTypes.InsEnergyCons;
	stSqlComandDataTMP.bWaitForDataReturn:=FALSE;
	
	sFormat := 'INSERT INTO `ProductionConsumption_Energy` (`IdLineStation`, `CounterValue`, `ValueUnit`) VALUES ( %d, %.3f, $'kWh$')';
	fbFormatStr2(pFormatString := ADR(sFormat),
			arg1:= F_DINT(stRetDataLineStation.IdStacji),
			arg2:= F_REAL(rActEnergyConsumption),
			pDstString := ADR(stSqlComandDataTMP.sCmdExpression), nDstSize := SIZEOF(stSqlComandDataTMP.sCmdExpression));
	stSqlComandDataTMP.pReturnedData := 0;
	stSqlComandDataTMP.uiReturnedDataSize := 0;	
	IF I_SqlCore <> 0 THEN
		m_SqlInsEnergyConsumption := I_SqlCore.mAddCmdToQueue(ADR(stSqlComandDataTMP));
	END_IF
ELSE
	m_SqlInsEnergyConsumption := FALSE;
END_IF
END_METHOD

// Zapis do DB danych rozszerzonych operacji - jeśli rozkaz dodany do kolejki zwraca TRUE, jeśli nie FALSE
METHOD m_SqlInsertExtendedData : BOOL		
VAR_INPUT
	pParameters: POINTER TO BYTE;				// Wskaźnik na tablicę elementów typu PIM_ExtDataRow
	uiArraySize: UINT;							// Rozmiar tablicy parametrów (może być pojedyncza zmienna)
END_VAR
VAR
	pExtData: POINTER TO stPIM_ExtDataRow;
	i:UINT;
	uiLastIndex:UINT;
END_VAR
uiLastIndex := uiArraySize/ SIZEOF(stPIM_ExtDataRow);
IF pParameters <> 0 AND uiArraySize > 0 AND uiLastIndex > 0 AND liLPartStatusId <> 0 THEN		// Zabezpieczenie przed brakiem danych wejściowych
	stSqlComandDataTMP.sCmdExpression := 'INSERT INTO `ProductionMachinePartParams` (`IdPartStatus`,`Name`,`Value`) VALUES';
	pExtData := pParameters;
	FOR i:=1 TO uiLastIndex DO		// Dodanie do stringa wartości
		IF i = uiLastIndex THEN		// Ostatnia wartość bez przecinka
			fbFormatStr(sFormat:= ' (%d,$'%s$',$'%s$')',arg1 := F_LINT(in:=liLPartStatusId), arg2 := F_STRINGEx(pExtData^.sName), arg3 := F_STRINGEx(pExtData^.sValue));
		ELSE
			fbFormatStr(sFormat:= ' (%d,$'%s$',$'%s$'),',arg1 := F_LINT(in:=liLPartStatusId), arg2 := F_STRINGEx(pExtData^.sName), arg3 := F_STRINGEx(pExtData^.sValue));		
			pExtData := pExtData + SIZEOF(stPIM_ExtDataRow);		// Przejście na kolejny indeks w tablicy
		END_IF
		CONCAT2(pSrcString1 := ADR(stSqlComandDataTMP.sCmdExpression), pSrcString2 := ADR(fbFormatStr.sOut), pDstString := ADR(stSqlComandDataTMP.sCmdExpression), nDstSize:= SIZEOF(stSqlComandDataTMP.sCmdExpression));
	END_FOR
	stSqlComandDataTMP.nCmdState:= nSQL_CmdExecState.New;
	stSqlComandDataTMP.nCmdType:=nSQL_CmdTypes.InsExtendedData;
	stSqlComandDataTMP.bWaitForDataReturn:=FALSE;
	stSqlComandDataTMP.pReturnedData := 0;
	stSqlComandDataTMP.uiReturnedDataSize := 0;
	IF I_SqlCore <> 0 THEN
  		m_SqlInsertExtendedData := I_SqlCore.mAddCmdToQueue(ADR(stSqlComandDataTMP));
	END_IF
ELSE
	m_SqlInsertExtendedData := FALSE;
END_IF
END_METHOD

// Zapis do DB parametrów maszyny przypisanych do aktualnego komponentu - gdy rozkaz zostanie wykonany zwraca TRUE
METHOD m_SqlInsMachineParamsData : BOOL
VAR_INPUT
	pParamsData: POINTER TO BYTE;		// Wskaźnik do bloku parametrów maszyny
	uiParamsDataSize: UINT;				// ROzmiar bloku danych parametrów maszyny
	wCrcSumOfParameters:WORD:= 0;
END_VAR
VAR_OUTPUT
	bProcessing:BOOL;					// Przetwarzanie rozkazu trwa (rozkaz dodany do kolejki)
	bResultOK:BOOL;						// Wynik wykonania rozkazu (do sprawdzenia gdy metoda zwróci TRUE)
	diParamsId:DINT;					// Id parametrów w DB
END_VAR
VAR
	sStringTMP:STRING(2000);
	iCRC16sum: INT;
END_VAR

// Sprawdzenie danych wejściowych - jeśli błędne przerwij procedure
IF pParamsData = 0 OR uiParamsDataSize = 0 OR stRetDataLineStation.IdStacji = 0 THEN 
	nErrorID:=nPIM_ErrorCodes.ProgramError;
	RETURN;
END_IF

// Rezerwacja struktury danych dla zapytania
IF NOT bReturnDataBusy OR bReturnDataReserved_InsMachParams THEN
	IF NOT bCmdSended THEN	// Przygotowanie danych do zapytania
		stSqlComandData.nCmdState:= nSQL_CmdExecState.New;
		stSqlComandData.nCmdType:=nSQL_CmdTypes.InsMachineParams;
		stSqlComandData.byExecutingNodeNb:=0;
		stSqlComandData.bWaitForDataReturn:=TRUE;
		
		IF wCrcSumOfParameters <> 0 THEN
			iCRC16sum := WORD_TO_INT(wCrcSumOfParameters);
		ELSE
			iCRC16sum := WORD_TO_INT(F_DATA_TO_CRC16_CCITT(pData := pParamsData, cbData := uiParamsDataSize, crc:= 0));
		END_IF
		fDataToHexStr(pData := pParamsData, uiDataSize := uiParamsDataSize, pStr := ADR(sStringTMP), uiStrSize := SIZEOF(sStringTMP));
		
		sFormat := 'UPDATE [dbo].[ProductionMachineParameters] SET Active = 0 WHERE IdLineStation = %d AND MachineNumber = %d AND IdComposedPart = %d DECLARE @ID_INSERTED TABLE (Id INT) INSERT INTO [dbo].[ProductionMachineParameters] (IdLineStation, MachineNumber, IdComposedPart,ParamsData,CRC_Sum,ParamsSizeInBytes) OUTPUT INSERTED.ID INTO @ID_INSERTED VALUES (%d, %d, %d, CAST( '; 
		fbFormatStr2(pFormatString := ADR(sFormat),
			arg1:= F_DINT(stRetDataLineStation.IdStacji),
			arg2:= F_INT(iMachineNumber),
			arg3:= F_LINT(stRetDataLineStation.IdOutComposedPart),
			arg4:= F_DINT(stRetDataLineStation.IdStacji),
			arg5:= F_INT(iMachineNumber),
			arg6:= F_LINT(stRetDataLineStation.IdOutComposedPart),
			pDstString := ADR(stSqlComandData.sCmdExpression), nDstSize := SIZEOF(stSqlComandData.sCmdExpression));
		CONCAT2(pSrcString1 := ADR(stSqlComandData.sCmdExpression), pSrcString2 := ADR(sStringTMP), pDstString :=ADR(stSqlComandData.sCmdExpression), nDstSize := SIZEOF(stSqlComandData.sCmdExpression));
		sFormat:= ' AS VARBINARY(%d)), %d,%d) SELECT Id FROM @ID_INSERTED';
		fbFormatStr2(pFormatString := ADR(sFormat),
			arg1:= F_UINT(uiParamsDataSize),
			arg2:= F_INT(iCRC16sum),
			arg3:= F_UINT(uiParamsDataSize),
			pDstString := ADR(sStringTMP), nDstSize := SIZEOF(sStringTMP));
		CONCAT2(pSrcString1 := ADR(stSqlComandData.sCmdExpression), pSrcString2 := ADR(sStringTMP), pDstString :=ADR(stSqlComandData.sCmdExpression), nDstSize := SIZEOF(stSqlComandData.sCmdExpression));	
		
